# B&R Automation Studio project ProjectOrionBms
Automation Studio 4.12.6.106; technology packages: mapp 5.24.1, mappView 5.24.1

## Configuration Config1

### Task classes (Cpu.sw)
```
Cyclic#1:
  INS <- INS.INS.prg
Cyclic#2:
  AMS_CAN <- AMS_and_Shunt.CAN.AMS_CAN.prg
  INV_CAN <- Inverters.CAN.CAN.prg
Cyclic#3:
  INV_CTRL <- Inverters.Control.Control.prg
Cyclic#4:
  INV_SM <- Inverters.Inv_statemachine.Inv_statemachine.prg
  SENSORS <- Sensors.Sensors.prg
  ACTUATORS <- Actuators.Output.prg
  DASHBOARD <- Dashboard.Dashboard.prg
  COOLING <- CoolingSystem.COOLING.prg
Cyclic#5:
  Simulation <- Inverters.Simulation.Simulation.prg [disabled]
  AMS_CTRL <- AMS_and_Shunt.AMS.prg
  SC <- SC.SafetyChain.prg
  SM <- SM.StateMachine.prg
  SENSOR_NET <- SensorNet.globalSensorNet.prg [disabled]
  ALARM_MAN <- Misc.AlarmManagement.AlarmManagement.prg
Cyclic#6:
  sampleST <- Misc.DataLogging.sampleST.prg [disabled]
  DATALOG <- Misc.DataLogging.DataLog.prg
Binaries: TCData, udbdef, mvLoader, arsvcreg, OpcUaMap, ashwac, Role, ashwd, arconfig, sysconf, iomap, User, asfw, Config_1, Config, Config_2, Config_3, Acp10map, acp10cfg
Libraries: runtime, astime, standard, operator, AsIecCon, AsIODiag, brsystem, asstring, ArCan, brdkSIM, brdkUSB, AsIO, AsBrStr, sys_lib, FileIO, AsUSB, DataObj, brdkSTR, MpAlarmX, MpBase, MpData, NcGlobal, MpRecipe, sduVikings, MTTypes, dvframe, MTFilter, areventlog
```

### Config.mpalarmxcore - X90CP174_48_00/mappServices/Config.mpalarmxcore
```
Element gAlarmXCore (Type=mpalarmxcore)
  mapp.AlarmX.Core.Configuration:
    [0]:
      Name = steeringAngleSensorDisconnected
      Message = Steering angle sensor disconnected
      Behavior = LevelMonitoring
        Acknowledge = 0
        Monitoring:
          MonitoredPV = ::gSteeringAngle.status.disconnected
          HighLimitEnable = Static
            Limit = 0.5
    [1]:
      Name = steeringAngleOutOfRange
      Message = Steering angle sensor values out of range
      Behavior = LevelMonitoring
        Acknowledge = 0
        Monitoring:
          MonitoredPV = ::gSteeringAngle.status.errorOutOfRange
          LowLimitEnable = Static
          HighLimitEnable = Static
            Limit = 0.5
    [2]:
      Name = brakePressureRearOutOfRange
      Message = Brake pressure rear {&LimitText}
      Behavior = LevelMonitoring
        Acknowledge = 0
        Monitoring:
          MonitoredPV = ::gBraking.inputs.ai_brakePressureRear
          LowLimitEnable = Dynamic
            LimitPV = ::SENSORS:brakingPedalConstants.rearWarningLimitMin
            LimitText = under low limit. 
            LowLowLimitEnable = Dynamic
              LimitPV = ::SENSORS:brakingPedalConstants.rearWarningLimitMinMin
              LimitText = under low low limit. 
          HighLimitEnable = Dynamic
            LimitPV = ::SENSORS:brakingPedalConstants.rearWarningLimitMax
            LimitText = over high limit. 
            HighHighLimitEnable = Dynamic
              LimitPV = ::SENSORS:brakingPedalConstants.rearWarningLimitMaxMax
              LimitText = over high high limit. 
    [3]:
      Name = brakePressureFrontOutOfRange
      Message = Brake pressure front {&LimitText}
      Behavior = LevelMonitoring
        Acknowledge = 0
        Monitoring:
          MonitoredPV = ::gBraking.inputs.ai_brakePressureFront
          LowLimitEnable = Dynamic
            LimitPV = ::SENSORS:brakingPedalConstants.frontWarningLimitMin
            LimitText = under low limit.
            LowLowLimitEnable = Dynamic
              LimitPV = ::SENSORS:brakingPedalConstants.frontWarningLimitMinMin
              LimitText = under low low limit.
          HighLimitEnable = Dynamic
            LimitPV = ::SENSORS:brakingPedalConstants.frontWarningLimitMax
            LimitText = over high limit.
            HighHighLimitEnable = Dynamic
              LimitPV = ::SENSORS:brakingPedalConstants.frontWarningLimitMaxMax
              LimitText = over high high limit.
    [4]:
      Name = torquePedalError1
      Message = Torque pedal sensor 1 out of range
      Behavior = LevelMonitoring
        Acknowledge = 0
        Monitoring:
          MonitoredPV = ::gTorqueSensor.inputs.torque1
          LowLimitEnable = Dynamic
            LimitPV = ::SENSORS:torquePedalConstants.lowLimit1
          HighLimitEnable = Dynamic
            LimitPV = ::SENSORS:torquePedalConstants..highLimit1
    [5]:
      Name = torquePedalError2
      Message = Torque pedal sensor 2 out of range
      Behavior = LevelMonitoring
        Acknowledge = 0
        Monitoring:
          MonitoredPV = ::gTorqueSensor.inputs.torque2
          LowLimitEnable = Dynamic
            LimitPV = ::SENSORS:torquePedalConstants.lowLimit2
          HighLimitEnable = Dynamic
            LimitPV = ::SENSORS:torquePedalConstants.highLimit2
    [6]:
      Name = PowerLimitWarning_fix
      Message = Warning! Power usage close to limit
      Behavior = LevelMonitoring
        Recording:
          InactiveToActive = FALSE
          UnacknowledgedToAcknowledged = FALSE
        Monitoring:
          MonitoredPV = ::gShunt.data.actPowerKW
          Exclusive = FALSE
          HighLimitEnable = Dynamic
            LimitPV = 
            LimitText = Warning! Power limit high
    [7]:
      Name = PowerLimitError_fix
      Message = Error! Power limit exceeded!
      Behavior = LevelMonitoring
        Recording:
          InactiveToActive = FALSE
          UnacknowledgedToAcknowledged = FALSE
        Monitoring:
          MonitoredPV = ::gShunt.data.actPowerKW
          HighLimitEnable = Dynamic
            LimitPV = 
            LimitText = 
    [8]:
      Name = coolingSystemManual
      Message = Cooling system on manual mode
      Behavior = LevelMonitoring
        Acknowledge = 0
        ReactionUntilAcknowledged = FALSE
        Recording:
          InactiveToActive = FALSE
          UnacknowledgedToAcknowledged = FALSE
        Monitoring:
          MonitoredPV = ::gCooling[0].cmd.manualMode
          HighLimitEnable = Static
            Limit = 0.1
    [9]:
      Name = stateChangeTimeout
      Message = State Machine never received confirmation and had a timeout
      Behavior = LevelMonitoring
        Recording:
          InactiveToActive = FALSE
          UnacknowledgedToAcknowledged = FALSE
        Monitoring:
          MonitoredPV = ::gStateMachine.status.stateChangeTimeout
          HighLimitEnable = Static
            Limit = 0.5
    [10]:
      Name = tractionControlDisabled
      Message = Traction Control not enabled
      Behavior = LevelMonitoring
        Acknowledge = 0
        ReactionUntilAcknowledged = FALSE
        Recording:
          InactiveToActive = FALSE
          UnacknowledgedToAcknowledged = FALSE
        Monitoring:
          MonitoredPV = ::gInverters.cmd.enableTractionControl
          LowLimitEnable = Static
            Limit = 0.5
    [11]:
      Name = torqueVectoringDisabled
      Message = Torque Vectoring not enabled
      Behavior = LevelMonitoring
        Acknowledge = 0
        ReactionUntilAcknowledged = FALSE
        Recording:
          InactiveToActive = FALSE
          UnacknowledgedToAcknowledged = FALSE
        Monitoring:
          MonitoredPV = ::gInverters.cmd.enableTorqueVectoring
          LowLimitEnable = Static
            Limit = 0.5
    [12]:
      Name = powerLimiterDisabled
      Message = Power Limiter not enabled
      Behavior = LevelMonitoring
        Acknowledge = 0
        Monitoring:
          MonitoredPV = ::gInverters.cmd.enablePowerLimiter
          LowLimitEnable = Static
            Limit = 0.5
    [13]:
      Name = regenBrakingDisabled
      Message = Regenerative Braking not enabled
      Behavior = LevelMonitoring
        Acknowledge = 0
        Monitoring:
          MonitoredPV = ::gInverters.cmd.enableRegenerativeBraking
          LowLimitEnable = Static
            Limit = 0.5
    [14]:
      Name = inverter1disabled
      Message = Inverter 1 disabled
      Behavior = LevelMonitoring
        Acknowledge = 0
        Monitoring:
          MonitoredPV = ::gInverters.inverter[0].status.inverterEnabled
          LowLimitEnable = Static
            Limit = 0.5
    [15]:
      Name = inverter2disabled
      Message = Inverter 2 disabled
      Behavior = LevelMonitoring
        Acknowledge = 0
        Monitoring:
          MonitoredPV = ::gInverters.inverter[1].status.inverterEnabled
          LowLimitEnable = Static
            Limit = 0.5
    [16]:
      Name = inverter3disabled
      Message = Inverter 3 disabled
      Behavior = LevelMonitoring
        Acknowledge = 0
        Monitoring:
          MonitoredPV = ::gInverters.inverter[2].status.inverterEnabled
          LowLimitEnable = Static
            Limit = 0.5
    [17]:
      Name = inverter4disabled
      Message = Inverter 4 disabled
      Behavior = LevelMonitoring
        Acknowledge = 0
        Monitoring:
          MonitoredPV = ::gInverters.inverter[3].status.inverterEnabled
          LowLimitEnable = Static
            Limit = 0.5
    [18]:
      Name = torqueLimiting
      Message = Torque Limiting is active
      Behavior = LevelMonitoring
        Acknowledge = 0
        Recording:
          InactiveToActive = FALSE
          UnacknowledgedToAcknowledged = FALSE
        Monitoring:
          MonitoredPV = ::gInverters.cmd.enableTorqueLimiter
          HighLimitEnable = Static
            Limit = 0.5
    [19]:
      Name = inverter1ErrorDiagnostics
      Message = Inverter 1 - Error {&inverter1ErrorDiag}
      Behavior = LevelMonitoring
        Monitoring:
          MonitoredPV = ::gInverters.inverter[0].inputs.com_errorDiagnostics
          HighLimitEnable = Static
            Limit = 0.5
    [20]:
      Name = inverter2ErrorDiagnostics
      Message = Inverter 2 - Error {&inverter2ErrorDiag}
      Behavior = LevelMonitoring
        Monitoring:
          MonitoredPV = ::gInverters.inverter[1].inputs.com_errorDiagnostics
          HighLimitEnable = Static
            Limit = 0.5
    [21]:
      Name = inverter3ErrorDiagnostics
      Message = Inverter 3 - Error {&inverter3ErrorDiag}
      Behavior = LevelMonitoring
        Monitoring:
          MonitoredPV = ::gInverters.inverter[2].inputs.com_errorDiagnostics
          HighLimitEnable = Static
            Limit = 0.5
    [22]:
      Name = inverter4ErrorDiagnostics
      Message = Inverter 4 - Error {&inverter4ErrorDiag}
      Behavior = LevelMonitoring
        Monitoring:
          MonitoredPV = ::gInverters.inverter[3].inputs.com_errorDiagnostics
          HighLimitEnable = Static
            Limit = 0.5
    [23]:
      Name = amsUnderVoltage
      Message = AMS Error - Cell voltage too low
      Behavior = LevelMonitoring
        Monitoring:
          MonitoredPV = ::gAMS.status.error.lowVoltage
          HighLimitEnable = Static
            Limit = 0.5
    [24]:
      Name = amsOverVoltage
      Message = AMS Error - Cell voltage too high
      Behavior = LevelMonitoring
        Monitoring:
          MonitoredPV = ::gAMS.status.error.highVoltage
          HighLimitEnable = Static
            Limit = 0.5
    [25]:
      Name = amsUnderTemperature
      Message = AMS Error - Cell temperature too low
      Behavior = LevelMonitoring
        Monitoring:
          MonitoredPV = ::gAMS.status.error.lowTemp
          HighLimitEnable = Static
            Limit = 0.5
    [26]:
      Name = amsOverTemperature
      Message = AMS Error - Cell temperature too high
      Behavior = LevelMonitoring
        Monitoring:
          MonitoredPV = ::gAMS.status.error.highTemp
          HighLimitEnable = Static
            Limit = 0.5
    [27]:
      Name = amsCommunicationErrorLTC
      Message = AMS Error - LTC6813 communication error
      Behavior = LevelMonitoring
        Monitoring:
          MonitoredPV = ::gAMS.status.error.ltc6813Com
          HighLimitEnable = Static
            Limit = 0.5
    [28]:
      Name = amsCommunicationErrorShunt
      Message = AMS Error - Shunt communication error
      Behavior = LevelMonitoring
        Monitoring:
          MonitoredPV = ::gAMS.status.error.shuntCom
          HighLimitEnable = Static
            Limit = 0.5
    [29]:
      Name = amsOpenSc
      Message = AMS Error - Unable to open safety circuit
      Behavior = LevelMonitoring
        Monitoring:
          MonitoredPV = ::gAMS.status.error.openSc
          HighLimitEnable = Static
            Limit = 0.5
    [30]:
      Name = amsCloseSc
      Message = AMS Error - Unable to close safety circuit
      Behavior = LevelMonitoring
        Monitoring:
          MonitoredPV = ::gAMS.status.error.closeSc
          HighLimitEnable = Static
            Limit = 0.5
    [31]:
      Name = amsOpenAirMinusError
      Message = AMS Error - 
Unable to open AIR- relay
      Behavior = LevelMonitoring
        Monitoring:
          MonitoredPV = ::gAMS.status.error.openAirMinus
          HighLimitEnable = Static
            Limit = 0.5
    [32]:
      Name = amsCloseAirMinusError
      Message = AMS Error - Unable to close AIR- relay
      Behavior = LevelMonitoring
        Monitoring:
          MonitoredPV = ::gAMS.status.error.closeAirMinus
          HighLimitEnable = Static
            Limit = 0.5
    [33]:
      Name = amsOpenAirPlusError
      Message = AMS Error - Unable to open AIR+ relay



      Behavior = LevelMonitoring
        Monitoring:
          MonitoredPV = ::gAMS.status.error.openAirPlus
          HighLimitEnable = Static
            Limit = 0.5
    [34]:
      Name = amsCloseAirPlusError
      Message = AMS Error - 
Unable to close AIR+ relay
      Behavior = LevelMonitoring
        Monitoring:
          MonitoredPV = ::gAMS.status.error.closeAirPlus
          HighLimitEnable = Static
            Limit = 0.5
    [35]:
      Name = amsOpenPreError
      Message = AMS Error - 
Unable to open precharge relay
      Behavior = LevelMonitoring
        Monitoring:
          MonitoredPV = ::gAMS.status.error.openPrePlus
          HighLimitEnable = Static
            Limit = 0.5
    [36]:
      Name = amsClosePreError
      Message = AMS Error - Unable to close precharge relay
      Behavior = LevelMonitoring
        Monitoring:
          MonitoredPV = ::gAMS.status.error.closePrePlus
          HighLimitEnable = Static
            Limit = 0.5
    [37]:
      Name = amsPrechargeTimeout
      Message = AMS Error - Precharge timeout
      Behavior = LevelMonitoring
        Monitoring:
          MonitoredPV = ::gAMS.status.error.preTimeout
          HighLimitEnable = Static
            Limit = 0.5
    [38]:
      Name = amsUnexpectedChargingRate
      Message = AMS Error - Unexpected Charge Rate
      Behavior = LevelMonitoring
        Monitoring:
          MonitoredPV = ::gAMS.status.error.unexpectedChargeRate
          HighLimitEnable = Static
            Limit = 0.5
    [39]:
      Name = amsUnexpectedTsCurrent
      Message = AMS Error - Unexpected TS Current
      Behavior = LevelMonitoring
        Monitoring:
          MonitoredPV = ::gAMS.status.error.unexpectedTsCurrent
          HighLimitEnable = Static
            Limit = 0.5
    [40]:
      Name = amsBankCountMismatch
      Message = AMS Error - The specified bank count from the Car does not match the meassured cells by the AMS
      Behavior = LevelMonitoring
        Monitoring:
          MonitoredPV = ::gAMS.status.error.bankCountMismatch
          HighLimitEnable = Static
            Limit = 0.5
    [41]:
      Name = amsScBroken
      Message = AMS Error - SC Broken
      Behavior = LevelMonitoring
        Monitoring:
          MonitoredPV = ::gAMS.status.error.scBroken
          HighLimitEnable = Static
            Limit = 0.5
    [42]:
      Name = amsUnfitChargingVoltage
      Message = AMS Error - Unfit Charge Voltage
      Behavior = LevelMonitoring
        Monitoring:
          MonitoredPV = ::gAMS.status.error.unexpectedChargeRate
          HighLimitEnable = Static
            Limit = 0.5
    [43]:
      Name = amsMonitorError
      Message = AMS Error - Monitor Error
      Behavior = LevelMonitoring
        Monitoring:
          MonitoredPV = ::gAMS.status.error.monitorError
          HighLimitEnable = Static
            Limit = 0.5
    [44]:
      Name = amsRelayFailed
      Message = AMS Error - Relay Failed
      Behavior = LevelMonitoring
        Monitoring:
          MonitoredPV = ::gAMS.status.error.relayFailed
          HighLimitEnable = Static
            Limit = 0.5
    [45]:
      Name = chargingCurrentWarning_fix
      Message = Charging Current Warning
      Behavior = LevelMonitoring
        Monitoring:
          MonitoredPV = 
          HighLimitEnable = Static
            Limit = 0.5
    [46]:
      Name = dashboardDisconnection
      Message = Dashboard Error - Disconnected
      Behavior = LevelMonitoring
        Acknowledge = 0
        Monitoring:
          MonitoredPV = ::gDashboard.status.DashboardDisconnected
          HighLimitEnable = Static
            Limit = 0.5
    [47]:
      Name = AMSDisconnection
      Message = AMS Error - Disconnected
      Behavior = LevelMonitoring
        Acknowledge = 0
        Monitoring:
          MonitoredPV = gAMS.status.disconnected
          HighLimitEnable = Static
            Limit = 0.5
    [48]:
      Name = RTDSDisconnection
      Message = RTDS Error - Disconnected
      Behavior = LevelMonitoring
        Acknowledge = 0
        Monitoring:
          MonitoredPV = gRTDS.status.RTDS_Disconnected
          HighLimitEnable = Static
            Limit = 0.5
    [49]:
      Name = Pump1Disconnection
      Message = Pump 1 Error - Disconnected
      Behavior = LevelMonitoring
        Acknowledge = 0
        Monitoring:
          MonitoredPV = gCooling.status.error[0]
          HighLimitEnable = Static
            Limit = 0.5
    [50]:
      Name = Pump2Disconnection
      Message = Pump 2 Error - Disconnected
      Behavior = LevelMonitoring
        Acknowledge = 0
        Monitoring:
          MonitoredPV = gCooling.status.error[1]
          HighLimitEnable = Static
            Limit = 0.5
    [51]:
      Name = LowVoltageBatteryLow
      Message = Warning! LV battery low 
      Behavior = LevelMonitoring
        Acknowledge = 0
        Monitoring:
          MonitoredPV = gLowVoltageBattery.status.empty
          HighLimitEnable = Static
            Limit = 0.5
    [52]:
      Name = inverter1Disconnected
      Message = Inverter 1 disconnected
      Behavior = LevelMonitoring
        Monitoring:
          MonitoredPV = ::gInverters.inverter[0].status.inverterDisconnected
          HighLimitEnable = Static
            Limit = 0.5
    [53]:
      Name = inverter2Disconnected
      Message = Inverter 2 disconnected
      Behavior = LevelMonitoring
        Acknowledge = 0
        Monitoring:
          MonitoredPV = ::gInverters.inverter[1].status.inverterDisconnected
          HighLimitEnable = Static
            Limit = 0.5
    [54]:
      Name = inverter3Disconnected
      Message = Inverter 3 disconnected
      Behavior = LevelMonitoring
        Acknowledge = 0
        Monitoring:
          MonitoredPV = ::gInverters.inverter[2].status.inverterDisconnected
          HighLimitEnable = Static
            Limit = 0.5
    [55]:
      Name = inverter4Disconnected
      Message = Inverter 4 disconnected
      Behavior = LevelMonitoring
        Acknowledge = 0
        Monitoring:
          MonitoredPV = ::gInverters.inverter[3].status.inverterDisconnected
          HighLimitEnable = Static
            Limit = 0.5
    [56]:
      Name = dataloggingInactive
      Message = Datalogging disabled
      Behavior = LevelMonitoring
        Monitoring:
          MonitoredPV = ::gDataLogging.status.dataloggingActive
          HighLimitEnable = Static
            Limit = 0.5
    [57]:
      Name = torquePedalPlausibilityError
      Message = Torque Pedal Plausibility Error
      Behavior = LevelMonitoring
        Monitoring:
          MonitoredPV = ::gTorqueSensor.status.plausibilityError
          HighLimitEnable = Static
            Limit = 0.5
    [58]:
      Name = shuntDisconnection
      Message = Shunt disconnected
      Behavior = LevelMonitoring
        Monitoring:
          MonitoredPV = ::gShunt.status.disconnected
          HighLimitEnable = Static
            Limit = 0.5
    [59]:
      Name = scBroken
      Message = SC Error - {&scErrorString}
      Behavior = DiscreteValueMonitoring
        ReactionUntilAcknowledged = FALSE
        Monitoring:
          MonitoredPV = ::gSafetyChain.status.scErrorIndex
          TriggerValues:
            [0] = 1
            [1] = 2
            [2] = 3
            [3] = 4
            [4] = 5
            [5] = 6
            [6] = 7
            [7] = 8
            [8] = 9
            [9] = 10
            [10] = 11
            [11] = 12
            [12] = 13
            [13] = 14
            [14] = 15
            [15] = 16
            [16] = 17
            [17] = 18
            [18] = 19
            [19] = 20
            [20] = 21
            [21] = 22
            [22] = 
    [60]:
      Name = inverterHighTemperature
      Message = Warning! Inverters are getting hot
      Behavior = LevelMonitoring
        Monitoring:
          MonitoredPV = ::gCooling.status.warningInverterHighTemp
          HighLimitEnable = Static
            Limit = 0.5
    [61]:
      Name = motorHighTemperature
      Message = Warning! Motors are getting hot
      Behavior = LevelMonitoring
        Monitoring:
          MonitoredPV = ::gCooling.status.warningMotorHighTemp
          HighLimitEnable = Static
            Limit = 0.5
    [62]:
      Name = orionBmsCommTimeout
      Message = Error! No Communication with Orion BMS
      Behavior = LevelMonitoring
        Monitoring:
          MonitoredPV = ::gORION.status.commTimeout
          HighLimitEnable = Static
            Limit = 0.5
  mapp.AlarmX.Core.Snippets:
    [0]:
      Key = inverter1ErrorDiag
      Value:
        PV = ::gInverters.inverter[0].inputs.com_errorDiagnostics
    [1]:
      Key = inverter2ErrorDiag
      Value:
        PV = ::gInverters.inverter[1].inputs.com_errorDiagnostics
    [2]:
      Key = inverter3ErrorDiag
      Value:
        PV = ::gInverters.inverter[2].inputs.com_errorDiagnostics
    [3]:
      Key = inverter4ErrorDiag
      Value:
        PV = ::gInverters.inverter[3].inputs.com_errorDiagnostics
    [4]:
      Key = scErrorString
      Value:
        PV = ::gSafetyChain.status.scErrorString
```

### Config_2.mpdatarecorder - X90CP174_48_00/mappServices/Config_2.mpdatarecorder
```
Element gDataRecorder (Type=mpdatarecorder)
```

### Config_3.mprecipexml - X90CP174_48_00/mappServices/Config_3.mprecipexml
```
Element gRecipeXml (Type=mprecipexml)
```

## Logical view

Binary libraries used (declarations not repeated): MpData 5.24.1

### Program Logical/Actuators/Output

#### Main.st
```iecst
PROGRAM _INIT
	(* Initialize outputs *)
	RtdsInit;

END_PROGRAM

PROGRAM _CYCLIC
	// Handle Ready-To-Drive-Sounds
	Rtds;

END_PROGRAM

PROGRAM _EXIT
	(* Insert code here *)

END_PROGRAM
```

### globalORION.typ
```iecst
TYPE
	gORION_state_ENUM :
		(
		INIT := 0,
		IDLE := 10,
		ENABLING_SC := 20,
		SC_ENABLED := 30,
		PRECHARGING := 40,
		PRECHARGING_DONE := 50,
		DRIVE_PRECHARGE_ACTIVE := 60,
		DRIVE := 70,
		ABORT := 80,
		ERROR := 90
		);
	gORION_relays_typ : 	STRUCT
		sdcEnable : BOOL;
		precharge : BOOL;
		airMinus : BOOL;
		airPlus : BOOL;
	END_STRUCT;
	gORION_typ : 	STRUCT
		state : gORION_state_ENUM;
		cmd : gORION_cmd_typ;
		status : gORION_status_typ;
		relays : gORION_relays_typ;
		data : gORION_data_typ;
	END_STRUCT;
	gORION_cmd_typ : 	STRUCT
		placeholder : USINT;
	END_STRUCT;
	gORION_status_typ : 	STRUCT
		sdcEnabled : BOOL;
		commTimeout : BOOL;
	END_STRUCT;
	gORION_data_typ : 	STRUCT
		packVoltage : REAL;
		prechargeLevel : REAL;
		carVoltage : REAL;
		maxPrechargeCurrent : REAL;
		chargeCurrent : REAL;
		outputCurrent : REAL;
		TON_counter : TON;
		CCL_KW : REAL;
		CCL : INT;
		DCL_KW : REAL;
		DCL : INT;
		rollingCounterOld : USINT;
		rollingCounter : USINT;
		packPower : REAL;
	END_STRUCT;
END_TYPE
```

### Program Logical/AMS_and_Shunt/AMS

#### Variables.var
```iecst
VAR
	k : UINT;
	j : USINT;
	i : UINT;
	tmpTemperatureMax : REAL;
	tmpTemperatureMin : REAL;
	tmpVoltageMax : REAL;
	tmpVoltageMin : REAL;
	tmpVoltage : REAL;
	TON_historySoc : TON;
	TON_historyCurrent : TON;
	TON_historyVoltage : TON;
	TON_historyPower : TON;
	powerHistoryInverval : TIME;
	currentHistoryInverval : TIME;
	voltageHistoryInverval : TIME;
	socHistoryInverval : TIME;
	powerWarningLimit : REAL;
	constant : constant_typ;
	CMD_ABORT : USINT := 0;
	CMD_ENABLE_SC : USINT := 1;
	CMD_ENABLE_TS : USINT := 2;
	CMD_ENABLE_DRIVE : USINT := 3;
	CMD_SET_BANK_COUNT : USINT := 5;
	CMD_SYNC_TIME : USINT := 6;
	inrushCurrentDetected : BOOL;
END_VAR
```

#### Main.st
```iecst
PROGRAM _INIT

	gAMS.data.outputCurrent := 0;
	gAMS.data.stateOfCharge := 0;
//	gAMS.data.totalPower 	:= 0;
//	gAMS.data.totalPowerMax := 0;  // Reset variable used to keep track of the maximum power used

	powerHistoryInverval 		:= T#10ms;
	currentHistoryInverval 		:= T#20ms;
	socHistoryInverval			:= T#500ms;
	voltageHistoryInverval  	:= T#100ms;
	gORION.data.TON_counter.PT	:= T#1s;

	constant.fullBatteryCapacityAh  := 12.5;
	constant.fullBatteryCapacitykWh := 6.475;

	constant.chargingCurrentMax := 12.5;
	gAMS.cmd.chargingPrescalerAmp := constant.chargingCurrentMax;

	gAMS.cmd.bankCount := 5;

	errorsInit_action;

END_PROGRAM

PROGRAM _CYCLIC

	states;
	orionErrorAction;
	error_action;

	gAMS.data.chargeCurrent := - gAMS.data.outputCurrent;

//	gAMS.data.batteryVoltage := gAMS.status.bank[0].bankVoltage + gAMS.status.bank[1].bankVoltage +
//								gAMS.status.bank[2].bankVoltage + gAMS.status.bank[3].bankVoltage +
//								gAMS.status.bank[4].bankVoltage;

	gAMS.cmd.chargingPrescalerPercent := LIMIT(0, REAL_TO_USINT((gAMS.cmd.chargingPrescalerAmp / constant.chargingCurrentMax) * 100), 100);

	powerMonitoring;

	(* Determine if AMS has an error or not *)
	gAMS.status.ok 	 := (NOT gAMS.status.disconnected) AND (NOT (gAMS.status.amsStateName = 'ERROR')) AND (NOT gAMS.status.hasError);
	gShunt.status.ok := NOT gShunt.status.disconnected;

//	gAMS.data.stateOfCharge := ((constant.fullBatteryCapacitykWh-gShunt.data.actPowerKWH) / constant.fullBatteryCapacitykWh) * 100.00;

	// Calculating the voltage of each bank
	FOR j := 0 TO BANK_COUNT-1 DO
		k := CELL_COUNT*j;
		tmpVoltage := 0;
		FOR i := 0 TO CELL_COUNT-1 DO
			// gAMS.status.bank[j].cellVoltage[i] := gAMS.status.pack.cellVoltage[i + k];
			tmpVoltage := tmpVoltage + gAMS.status.bank[j].cellVoltage[i];
		END_FOR;
		gAMS.status.bank[j].bankVoltage := tmpVoltage;
	END_FOR

	FOR j := 0 TO BANK_COUNT-1 DO
		// Max voltage
		tmpVoltageMax := 0;
		FOR i := 0 TO CELL_COUNT-1 DO
			IF gAMS.status.bank[j].cellVoltage[i] > tmpVoltageMax THEN
				tmpVoltageMax := gAMS.status.bank[j].cellVoltage[i];
			END_IF;
		END_FOR;
		gAMS.data.cellVoltageMax[j] := tmpVoltageMax;

		// Min voltage
		tmpVoltageMin := 10000;
		FOR i := 0 TO CELL_COUNT-1 DO
			IF gAMS.status.bank[j].cellVoltage[i] < tmpVoltageMin THEN
				tmpVoltageMin := gAMS.status.bank[j].cellVoltage[i];
			END_IF;
		END_FOR;
		gAMS.data.cellVoltageMin[j] := tmpVoltageMin;

		// Max temperature
		tmpTemperatureMax := 0;
		FOR i := 0 TO TEMPERATURE_COUNT-1 DO
			IF gAMS.status.bank[j].temperatures[i] > tmpTemperatureMax THEN
				tmpTemperatureMax := gAMS.status.bank[j].temperatures[i];
			END_IF;
		END_FOR;
		gAMS.data.bankTemperatureMax[j] := tmpTemperatureMax;

		// Min temperature
		tmpTemperatureMin := 10000;
		FOR i := 0 TO TEMPERATURE_COUNT-1 DO
			IF gAMS.status.bank[j].temperatures[i] < tmpTemperatureMin THEN
				tmpTemperatureMin := gAMS.status.bank[j].temperatures[i];
			END_IF;
		END_FOR;
		gAMS.data.bankTemperatureMin[j] := tmpTemperatureMin;

		// Max resistor temperature
		tmpTemperatureMax := 0;
		FOR i := 0 TO RESISTOR_COUNT-1 DO
			IF gAMS.status.bank[j].resistorTemperature[i] > tmpTemperatureMax THEN
				tmpTemperatureMax := gAMS.status.bank[j].resistorTemperature[i];
			END_IF;
		END_FOR;
		gAMS.data.bankResistorTemperatureMax[j] := tmpTemperatureMax;

		// Min temperature
		tmpTemperatureMin := 10000;
		FOR i := 0 TO RESISTOR_COUNT-1 DO
			IF gAMS.status.bank[j].resistorTemperature[i] < tmpTemperatureMin THEN
				tmpTemperatureMin := gAMS.status.bank[j].resistorTemperature[i];
			END_IF;
		END_FOR;
		gAMS.data.bankResistorTemperatureMin[j] := tmpTemperatureMin;

	END_FOR;

	history;

END_PROGRAM

PROGRAM _EXIT
	(* Insert code here *)

END_PROGRAM
```

#### powerMonitoring.st
```iecst
(* Keep track of the current power consumption and the maximum power *)
ACTION powerMonitoring:
	// Actual power
//	gAMS.data.totalPowerKW := gAMS.data.totalPower / 1000.00;

	// Maximum power
//	IF gAMS.data.totalPower > gAMS.data.totalPowerMax THEN
//		gAMS.data.totalPowerMax := gAMS.data.totalPower;
//		gAMS.data.totalPowerMaxKW := gAMS.data.totalPowerMax / 1000.00;
//	END_IF;

	IF gInverters.cmd.enablePowerLimiter THEN
//		powerWarningLimit := gInverters.data.powerLimitKW*0.9;
//		IF gAMS.data.totalPowerKW > 1 THEN
//			gAMS.status.highPowerWarning := powerWarningLimit 					<= gAMS.data.totalPowerKW;
//			gAMS.status.highPowerError   := gInverters.data.powerLimitKW 	<= gAMS.data.totalPowerKW;
//		END_IF;
	ELSE
		gAMS.status.highPowerWarning := FALSE;
		gAMS.status.highPowerError   := FALSE;
	END_IF;

END_ACTION
```

### Program Logical/AMS_and_Shunt/CAN/AMS_CAN (IEC)

#### Main.st
```iecst
PROGRAM _INIT
	(* Device *)
	deviceName 						:= 'IF9';
	(* Bus *)
	ArCanSetBaudrate_0.Baudrate 	:= 500000;
	(* Transmit *)
	ArCanSend_0.Frame.Format 		:= arCAN_11BIT;
	(* Receive *)
	ArCanReceive_0.Format 			:= arCAN_11BIT;
	ArCanReceive_0.QueueSize		:= 100;
	ArCanReceive_0.IDMask			:= arCAN_RECEIVE_ALL;

	communicationState := S_INIT;

	RX_CAN_ID_BASE 		:= 16#300;
	TX_CAN_ID_BASE 		:= 16#300;
	RX_ORION_ID_BASE	:= 16#400;
	TX_ORION_ID_BASE	:= 16#400;
	SHUNT_ID_BASE  		:= 16#500;

	NO_OF_BANKS := 4;
//	gAMS.status.error.dataFrameLost := FALSE;

END_PROGRAM

PROGRAM _CYCLIC

	CASE communicationState OF
		S_INIT:
			(* PLC is not simulated. It is run on an actual PLC *)
			IF NOT gIsSimulation THEN

				(* Configure CAN port *)
				ArCanSetBaudrate_0.DeviceName	:= deviceName;
				ArCanSetBaudrate_0.Execute 		:= TRUE;
				IF ArCanSetBaudrate_0.Done THEN
					communicationState 			:= S_INIT_TX;
				END_IF;
				IF ArCanSetBaudrate_0.Error THEN
					communicationState 			:= S_ERROR;
				END_IF;
			ELSE
				(* PLC is simulated. It is run in the simulator and no hardware is connnected *)
				communicationState 				:= S_IDLE;
			END_IF;

		S_INIT_TX: // Init Tx
			(* Configure send function block *)
			ArCanSend_0.Enable 			:= TRUE;
			ArCanSend_0.DeviceName 		:= deviceName;

			IF ArCanSend_0.Active THEN
				communicationState 		:= S_INIT_RX;
			END_IF;

			IF ArCanSend_0.Error THEN
				communicationState 		:= S_ERROR;
			END_IF;

		S_INIT_RX:	// Init Rx
			(* Configure receive function block *)
			ArCanReceive_0.Enable 		:= TRUE;
			ArCanReceive_0.DeviceName 	:= deviceName;

			IF ArCanReceive_0.Active THEN
				communicationState 		:= S_RUNNING;
			END_IF;

			IF ArCanReceive_0.Error THEN
				communicationState 		:= S_ERROR;
			END_IF

		S_RUNNING: // Running
			AMS_Send;		// Handle transmit task
			AMS_Receive;	// Handle receive task

		S_ERROR: // Error
			IF ArCanSend_0.Error THEN
				ArCanSend_0(Enable := FALSE);
				ArCanSend_0(Enable := TRUE);
			END_IF;

			IF ArCanReceive_0.Error THEN
				ArCanReceive_0(Enable := FALSE);
				ArCanReceive_0(Enable := TRUE);
			END_IF;

			IF (ArCanReceive_0.Error = FALSE) AND (ArCanSend_0.Error = FALSE) AND (ArCanSetBaudrate_0.Error = FALSE) THEN
				communicationState 		:= S_INIT;
			END_IF;
		S_IDLE: // Do nothing
	END_CASE

	IF NOT gIsSimulation THEN
		ArCanSetBaudrate_0();
		ArCanReceive_0();
		ArCanSend_0();
	END_IF;

//	gAMS.status.error.dataFrameLost := ArCanReceive_0.NumberOfLostFrames <> 0;

END_PROGRAM

PROGRAM _EXIT
	(* Insert code here *)

END_PROGRAM
```

### Program Logical/CoolingSystem/COOLING

#### Variables.var
```iecst
VAR
	COOLING_MODE_STATE : USINT := 0;
	pumpOffCurrent : UINT;
	pumpOnCurrent : UINT;
	i : USINT;
END_VAR
```

#### Main.st
```iecst
PROGRAM _INIT
	pumpOffCurrent := 1000;
	pumpOnCurrent  := 9500;
	gCooling.cmd.manualMode := FALSE;
	//gCooling.outputs.do_pump[1] := TRUE;
	FOR i := 0 TO 1 DO
		gCooling.outputs.do_pump[i] 	:= TRUE;
		gCooling.outputs.do_fan[i] 		:= TRUE;
		//gCooling.outputs.do_pump[i] 	:= FALSE;
		//gCooling.outputs.do_fan[i] 		:= FALSE;
	END_FOR

	gCooling.status.warningHighTemperature := FALSE;

	gCooling.cmd.inverterMaxTemp 	:= 60.0;
	gCooling.cmd.motorMaxTemp 		:= 100.0;
END_PROGRAM

PROGRAM _CYCLIC

	CASE COOLING_MODE_STATE OF
		0: // AUTO MODE
			IF gDashboard.inputs.di_button2 AND (gInverters.inverter[0].data.actualVelocityKmh = 0) THEN
	  			COOLING_MODE_STATE := 10;
			END_IF;
			IF gStateMachine.status.state = STATE_DRIVE THEN
				COOLING_MODE_STATE := 10;
			END_IF;
		10: // going to MANUAL MODE
			IF NOT gDashboard.inputs.di_button2 THEN
				gCooling.cmd.manualMode := TRUE;
				gCooling.outputs.do_pump[1] := TRUE;
				COOLING_MODE_STATE := 20;
			END_IF;

		20: // MANUAL MODE
			IF gDashboard.inputs.di_button2 AND (gInverters.inverter[0].data.actualVelocityKmh = 0) THEN
				COOLING_MODE_STATE := 30;
			END_IF;

		30:
			IF NOT gDashboard.inputs.di_button2 THEN
				gCooling.cmd.manualMode := FALSE;
				gCooling.outputs.do_pump[1] := FALSE;
				COOLING_MODE_STATE := 0;
			END_IF
	END_CASE;

	(* Convert analog temperature inputs to temperatures in degrees *)
	FOR i := 0 TO 1 DO
		(* Cooling System Temperature approximated via 4th order polynomium *)
		gCooling.data.coolingSysTemp[i] := EXPT(gCooling.inputs.ai_coolingTemp[i],2) + 0.004914 * gCooling.inputs.ai_coolingTemp[i] - 44.62;
	END_FOR

	// If cooling system is not in manual mode (its in automatic mode)
	IF NOT gCooling.cmd.manualMode THEN
		FOR i := 0 TO 1 DO
			//IF gCooling.outputs.do_pump[i] THEN
				//IF INT_TO_UINT(gCooling.inputs.im_pumpCurrent[i]) < pumpOffCurrent THEN
					// No current is being drawn
				//	gCooling.status.pumpState[i] := PUMP_STATE_NOT_CONNECTED;
				//ELSIF INT_TO_UINT(gCooling.inputs.im_pumpCurrent[i]) > pumpOffCurrent AND INT_TO_UINT(gCooling.inputs.im_pumpCurrent[i]) < pumpOnCurrent THEN
					// Not enough current is being drawn
				//	gCooling.status.pumpState[i] := PUMP_STATE_NO_WATER;
				//ELSE
			// Normal amount of current is being drawn
				IF gStateMachine.status.state = STATE_TRACTIVE THEN
					gCooling.status.pumpState[i] := PUMP_STATE_OK;
				ELSE
					gCooling.status.pumpState[i] := PUMP_STATE_NO_WATER; // Just to turn off when not in tractive
				END_IF;

				// Check if there is an error on the pump. If the pump state is not OK there is an error
				gCooling.status.pumpError[i] := gCooling.status.pumpState[i] <> PUMP_STATE_OK;

				// If there is an error turn OFF the pump. Otherwise keep it ON
				gCooling.outputs.do_pump[i] := NOT gCooling.status.pumpError[i];

			//END_IF

		END_FOR
	END_IF;

	// Enable fan when in STATE_DRIVE
	FOR i := 0 TO 1 DO
		gCooling.outputs.do_fan[i] := gStateMachine.status.state = STATE_DRIVE;
	END_FOR;

	// Evaluate if inverter or motors have high temperature errors
	gCooling.status.warningInverterHighTemp := MAX(gInverters.inverter[0].data.tempInverter, gInverters.inverter[1].data.tempInverter, gInverters.inverter[2].data.tempInverter, gInverters.inverter[3].data.tempInverter) > gCooling.cmd.inverterMaxTemp;
	gCooling.status.warningMotorHighTemp 	:= MAX(gInverters.inverter[0].data.tempMotor   , gInverters.inverter[1].data.tempMotor,    gInverters.inverter[2].data.tempMotor,    gInverters.inverter[3].data.tempMotor)    > gCooling.cmd.motorMaxTemp;

	// Evaluate if the cooling system is working properly.
	gCooling.status.ok := NOT gCooling.status.pumpError[0] AND NOT gCooling.status.pumpError[1];

	// Evaluate if the cooling system sees any temperature higher than allowed
	gCooling.status.warningHighTemperature := gCooling.status.warningInverterHighTemp OR gCooling.status.warningMotorHighTemp;
END_PROGRAM

PROGRAM _EXIT
	(* Insert code here *)

END_PROGRAM
```

### globalDashboard.var
```iecst
VAR
	gDashboard : gDashboard_typ;
END_VAR
```

### Program Logical/Dashboard/Dashboard/ledControl

#### ledDV.st
```iecst
(* Control the DV LED *)
ACTION ledDV:
	IF gStateMachine.status.state = STATE_INITIALIZE THEN
		gDashboard.outputs.do_ledDV := TRUE;
	ELSE
		gDashboard.outputs.do_ledDV := FALSE;
	END_IF;
END_ACTION
```

#### ledEBS.st
```iecst
(* Control the EBS LED *)
ACTION ledEBS:
	IF gStateMachine.status.state = STATE_INITIALIZE THEN
		gDashboard.outputs.do_ledEBS := TRUE;
	ELSE
		gDashboard.outputs.do_ledEBS := FALSE;
	END_IF;
END_ACTION
```

#### ledIMD.st
```iecst
(* Control the IMD LED *)
ACTION ledIMD:
	IF gStateMachine.status.state = STATE_INITIALIZE THEN
		gDashboard.outputs.do_ledIMD := TRUE;
	ELSE
		gDashboard.outputs.do_ledIMD := gAMS.status.error.imdError;
	END_IF;
END_ACTION
```

#### ledLV.st
```iecst
(* Control the LV LED *)
ACTION ledLV:

	IF gStateMachine.status.state = STATE_INITIALIZE THEN
		gDashboard.outputs.do_ledLV := FALSE;

	ELSE
		IF gLowVoltageBattery.status.empty THEN
			gDashboard.outputs.do_ledLV := TRUE;
		ELSE
			gDashboard.outputs.do_ledLV := FALSE;
		END_IF;

	END_IF;

END_ACTION
```

#### ledREADY.st
```iecst
(* Control the READY LED *)
ACTION ledREADY:
	IF gStateMachine.status.state = STATE_INITIALIZE THEN
		gDashboard.outputs.do_ledREADY := READY_ON;
	ELSE
		IF gStateMachine.status.state = STATE_DRIVE THEN
			gDashboard.outputs.do_ledREADY := READY_ON;
		ELSIF gStateMachine.status.readyForStateDrive THEN
			gDashboard.outputs.do_ledREADY := READY_FAST_BLINK;
		ELSIF gStateMachine.status.state = STATE_TRACTIVE THEN
			gDashboard.outputs.do_ledREADY := READY_SLOW_BLINK;
		ELSE
			gDashboard.outputs.do_ledREADY := READY_OFF;
		END_IF
	END_IF

	// Slow blink: State = TRACTIVE
	// Fast blink: State = TRACTIVE & gBraking.status.softBraking = TRUE & NOT gTorqueSensor.status.criticalError
	// On = DRIVE
	// Off : Else

END_ACTION
```

### Program Logical/Dashboard/Dashboard/Receive

#### receive_messages.st
```iecst
ACTION msg_0x050:
	gDashboard.inputs.di_buttonSafety		:= ArCanReceive_0.ReceivedFrame.Data[0].0;
	gDashboard.inputs.di_buttonTractive		:= ArCanReceive_0.ReceivedFrame.Data[0].1;
	gDashboard.inputs.di_buttonDrive		:= ArCanReceive_0.ReceivedFrame.Data[0].2;
	gDashboard.inputs.di_button1			:= ArCanReceive_0.ReceivedFrame.Data[0].3;
//
//	gDashboard.inputs.di_buttonDrive		:= ArCanReceive_0.ReceivedFrame.Data[0].3;
//	gDashboard.inputs.di_button1			:= ArCanReceive_0.ReceivedFrame.Data[0].2;
//
	gDashboard.inputs.di_button2			:= ArCanReceive_0.ReceivedFrame.Data[0].4;
	gDashboard.inputs.di_button3			:= ArCanReceive_0.ReceivedFrame.Data[0].5;
	gDashboard.inputs.di_button4			:= ArCanReceive_0.ReceivedFrame.Data[0].6;
END_ACTION

ACTION msg_0x051:
	gDashboard.status.statusIndex := BYTE_TO_USINT(ArCanReceive_0.ReceivedFrame.Data[0]);
END_ACTION

ACTION msg_0x052:
	(* Chagne driving mission *)
	CASE BYTE_TO_USINT(ArCanReceive_0.ReceivedFrame.Data[0]) OF
		MISSION_NONE: 		  gStateMachine.status.missionIndex := MISSION_NONE;
		MISSION_ACCELERATION: gStateMachine.status.missionIndex := MISSION_ACCELERATION;
		MISSION_SKIDPAD: 	  gStateMachine.status.missionIndex := MISSION_SKIDPAD;
		MISSION_SPRINT: 	  gStateMachine.status.missionIndex := MISSION_SPRINT;
		MISSION_ENDURANCE: 	  gStateMachine.status.missionIndex := MISSION_ENDURANCE;
		MISSION_BRAKE_TEST:	  gStateMachine.status.missionIndex := MISSION_BRAKE_TEST;
		MISSION_TESTING: 	  gStateMachine.status.missionIndex := MISSION_TESTING;
		ELSE	  			  gStateMachine.status.missionIndex := MISSION_NONE;
	END_CASE;
END_ACTION
```

### send_messages.st
```iecst
(*
Protocol specifications
https://gitlab.com/sdu-vikings/X/master-controller/-/wikis/Dashboard-CAN-Protocol
*)

ACTION msg_0x000:
	ArCanSend_0.Frame.ID 		  := TX_CAN_ID_BASE + 16#000; // CAN-ID
	ArCanSend_0.Frame.DataLength  := 6; 	 // Datalength

	speed 			:=	REAL_TO_INT(  gINS.data.actLonVelocity_kmh * 10.00 );
	soc 			:=	REAL_TO_INT(  gAMS.data.stateOfCharge * 10.00 );
	maxTemperature  := 	REAL_TO_UINT(MAX(gInverters.inverter[0].data.tempMotor, gInverters.inverter[1].data.tempMotor, gInverters.inverter[2].data.tempMotor, gInverters.inverter[3].data.tempMotor) * 10.00);

	memcpy(ADR(ArCanSend_0.Frame.Data[0]), ADR( speed 			), 2);
	memcpy(ADR(ArCanSend_0.Frame.Data[2]), ADR( soc 			), 2);
	memcpy(ADR(ArCanSend_0.Frame.Data[4]), ADR( maxTemperature	), 2);

END_ACTION

ACTION msg_0x001:
	ArCanSend_0.Frame.ID 		  := TX_CAN_ID_BASE+ 16#001; // CAN-ID
	ArCanSend_0.Frame.DataLength  := 4; 	 // Datalength

	memcpy(ADR(ArCanSend_0.Frame.Data[0]), ADR( gStateMachine.status.instructionIndex 	), 1);
	memcpy(ADR(ArCanSend_0.Frame.Data[1]), ADR( gStateMachine.status.state 				), 1);
	ArCanSend_0.Frame.Data[2].0 := gDashboard.outputs.com_error_Datalog;
	ArCanSend_0.Frame.Data[2].1 := gDashboard.outputs.com_error_SC;
	ArCanSend_0.Frame.Data[2].2 := gDashboard.outputs.com_error_Shunt;
	ArCanSend_0.Frame.Data[2].3 := gDashboard.outputs.com_error_AMS;
	ArCanSend_0.Frame.Data[2].4 := gDashboard.outputs.com_error_Dashboard;
	ArCanSend_0.Frame.Data[2].5 := gDashboard.outputs.com_error_3rd_Inv;
	ArCanSend_0.Frame.Data[2].6 := gDashboard.outputs.com_error_2nd_Inv;
	ArCanSend_0.Frame.Data[2].7 := gDashboard.outputs.com_error_1st_Inv;
	ArCanSend_0.Frame.Data[3].0 := gDashboard.outputs.com_error_0_Inv;
	ArCanSend_0.Frame.Data[3].1 := gDashboard.outputs.com_error_INS;
	ArCanSend_0.Frame.Data[3].2 := gDashboard.outputs.com_error_SteeringAngle;
	ArCanSend_0.Frame.Data[3].3 := gDashboard.outputs.com_error_BreakPressure_Front;
	ArCanSend_0.Frame.Data[3].4 := gDashboard.outputs.com_error_BreakPressure_Back;
	ArCanSend_0.Frame.Data[3].5 := gDashboard.outputs.com_error_TorquePedal;
	ArCanSend_0.Frame.Data[3].6 := gDashboard.outputs.com_error_TorquePedal_Plausi;
	ArCanSend_0.Frame.Data[3].7 := gDashboard.outputs.com_error_RTDS;
	ArCanSend_0.Frame.Data[4].0 := gDashboard.outputs.com_error_Cooling;
	ArCanSend_0.Frame.Data[4].1 := gDashboard.outputs.com_error_LV;
	ArCanSend_0.Frame.Data[4].2 := gDashboard.outputs.com_error_HighTemperature;

END_ACTION

ACTION msg_0x002:
	ArCanSend_0.Frame.ID 		  := TX_CAN_ID_BASE + 16#002; // CAN-ID
	ArCanSend_0.Frame.DataLength  := 2; 	 // Datalength

	ArCanSend_0.Frame.Data[0].0 := gDashboard.outputs.do_ledIMD;
	ArCanSend_0.Frame.Data[0].1 := gDashboard.outputs.do_ledAMS;
	ArCanSend_0.Frame.Data[0].2 := gDashboard.outputs.do_ledSC.0;
	ArCanSend_0.Frame.Data[0].3 := gDashboard.outputs.do_ledSC.1;
	ArCanSend_0.Frame.Data[0].4 := gDashboard.outputs.do_ledEBS;
	ArCanSend_0.Frame.Data[0].5 := gDashboard.outputs.do_ledDV;
	ArCanSend_0.Frame.Data[0].6 := gDashboard.outputs.do_ledREADY.0;
	ArCanSend_0.Frame.Data[0].7 := gDashboard.outputs.do_ledREADY.1;
	ArCanSend_0.Frame.Data[1].0 := gDashboard.outputs.do_ledLV;

END_ACTION

ACTION msg_0x003:
	ArCanSend_0.Frame.ID 		  := TX_CAN_ID_BASE + 16#003; // CAN-ID
	ArCanSend_0.Frame.DataLength := 6; 	 // Datalength

	memcpy(ADR(ArCanSend_0.Frame.Data[0]), ADR(gStateMachine.status.missionIndex), 1);

	ArCanSend_0.Frame.Data[1].0 := gInverters.cmd.enableTorqueVectoring;
	ArCanSend_0.Frame.Data[1].1 := gInverters.cmd.enableTractionControl;
	ArCanSend_0.Frame.Data[1].2 := gInverters.cmd.enablePowerLimiter;
	ArCanSend_0.Frame.Data[1].3 := gInverters.cmd.enableTorqueLimiter;
	//	ArCanSend_0.Frame.Data[1].4 := gInverters.cmd.enableLaunchProfile;
	ArCanSend_0.Frame.Data[1].5 := gInverters.cmd.enableRegenerativeBraking;
	ArCanSend_0.Frame.Data[1].6 := gInverters.status.regenerativeBrakingAvailable;
	torqueLimitNm  				:= REAL_TO_UINT(gInverters.data.torqueSetpointGain * 10.00);
	powerLimitKW  				:= REAL_TO_UINT(gInverters.data.powerLimitKW * 10.00);

	memcpy(ADR(ArCanSend_0.Frame.Data[2]), ADR(torqueLimitNm), 2);
	memcpy(ADR(ArCanSend_0.Frame.Data[4]), ADR(powerLimitKW), 2);
END_ACTION

ACTION msg_0x004:
	ArCanSend_0.Frame.ID 		  := TX_CAN_ID_BASE + 16#004; // CAN-ID
	ArCanSend_0.Frame.DataLength := 4; 	 // Datalength

	lvBatVoltage  		:= 	REAL_TO_UINT( gLowVoltageBattery.data.voltage * 10.00 );
	estimatedRange  	:=  REAL_TO_UINT( gINS.data.distEstimated * 10.00 );

	memcpy(ADR(ArCanSend_0.Frame.Data[0]), ADR( lvBatVoltage 	), 2);
	memcpy(ADR(ArCanSend_0.Frame.Data[2]), ADR( estimatedRange  ), 2);

END_ACTION
```

### Program Logical/INS/INS

#### Main.st
```iecst
PROGRAM _INIT
	// Enable serial communication
	Receiver.Commands.open_receive := TRUE;												(*enable Receiver by default*)

	(* Range Estimation *)
	MTFilterMovingAverage_0.Enable 		 := TRUE;
	MTFilterMovingAverage_0.WindowLength := 10;
	TON_rangEstTimer.PT 				 := T#10s;

	// Get cycle time
	RTInfo_0(enable := TRUE);
	cycletime := RTInfo_0.cycle_time / 1000; //[ms]

	gINS.data.distEstimated := 0;
END_PROGRAM

PROGRAM _CYCLIC

	// If the state is any of the 3 states used for receiving and decoding data mark the INS as ok
	// Otherwise mark it as not ok
	gINS.status.ok := Receiver.step = FRM_READ OR Receiver.step = FRM_COPY_RD_DATA OR Receiver.step = FRM_RBUF;

	// Handle communication
	CASE Receiver.step OF
		FRM_WAIT:	(*--- wait for command*)

			IF Receiver.Commands.open_receive = TRUE THEN								(*command for Receiver activation*)
				Receiver.step := FRM_OPEN;
			END_IF

			(*close will be requested in step FRM_RBUF*)

		FRM_OPEN:	(*--- open serial interface*)

			(*Parameters for FRM_xopen()*)
			Receiver.FRM_xopen_0.enable := TRUE;
			Receiver.FRM_xopen_0.device := ADR('IF6.ST1.IF4');							(*Devicename --> see your serial interface properties*)
			Receiver.FRM_xopen_0.mode := ADR('/PHY=RS232 /BD=115200 /DB=8 /PA=E /SB=1'); (*Modestring --> specifies the seria operation mode*)
			Receiver.FRM_xopen_0.config := ADR(Receiver.xopenConfig) ;					(*Additional Parameters, optional*)

			(*Additional Parameters for FRM_xopen()*)
			Receiver.xopenConfig.idle     := 10;								(*Idle time between two characters*)
			Receiver.xopenConfig.delimc   := 0;									(*activate two delimeters*)
			Receiver.xopenConfig.delim[0] := 0; 								(*e.g. CR - carridge return -> dec 13*)
			Receiver.xopenConfig.delim[1] := 0; 								(*e.g. LF - line feed -> dec 10*)
			Receiver.xopenConfig.tx_cnt   := 3;									(*number of transmit buffers*)
			Receiver.xopenConfig.rx_cnt   := 3; 								(*number of receive buffers*)
			Receiver.xopenConfig.tx_len   := 0; 								(*length of transmit buffers*)
			Receiver.xopenConfig.rx_len   := 44; 								(*lenght of receive buffers*)
			Receiver.xopenConfig.argc     := 0;									(*activate additional options*)
			Receiver.xopenConfig.argv     := 0;									(*parameters for additional options (check help)*)

			Receiver.FRM_xopen_0();												(*call the FRM_xopen() function*)

			IF Receiver.FRM_xopen_0.status = 0 THEN
				Receiver.step := FRM_READ;										(*Interface opend successfully --> next step*)
			ELSIF Receiver.FRM_xopen_0.status = BUSY THEN
				Receiver.step := FRM_OPEN;										(*operation not finished yet --> call again*)
			ELSE
				Receiver.step := FRM_ERROR;										(*function returned errorcode --> check help*)
			END_IF

		FRM_READ:	(*--- read data from serial interface*)
			Receiver.FRM_read_0.enable := TRUE;
			Receiver.FRM_read_0.ident := Receiver.FRM_xopen_0.ident;

			Receiver.FRM_read_0();												(*call the FRM_read() function*)

			IF Receiver.FRM_read_0.status = 0 THEN
				Receiver.step := FRM_COPY_RD_DATA;								(*system returned a valid data --> next step*)
			ELSIF Receiver.FRM_read_0.status = frmERR_NOINPUT THEN
				Receiver.step := FRM_READ;										(*no data available --> call again*)
			ELSIF Receiver.FRM_read_0.status = frmERR_INPUTERROR THEN
				Receiver.step := FRM_RBUF;										(*received Frame with defective characters, skip data*)
			ELSE
				Receiver.step := FRM_ERROR;										(*function returned errorcode --> check help*)
			END_IF

		FRM_COPY_RD_DATA: (*--- copy data out of the receive buffer*)
			memset(ADR(Receiver.receive_data),0,SIZEOF(Receiver.receive_data));			(*clear read_data buffer*)
			memcpy(ADR(Receiver.receive_data),Receiver.FRM_read_0.buffer,Receiver.FRM_read_0.buflng);     (*copy and evaluate read data*)
			checkMessageValidity;
			IF messageOk THEN
				extractInsData;
			END_IF;
			Receiver.step := FRM_RBUF;													(*release read buffer*)

		FRM_RBUF:	(*--- release readbuffer*)

			(*Parameters for FRM_rbuf()*)
			Receiver.FRM_rbuf_0.enable := TRUE;
			Receiver.FRM_rbuf_0.ident := Receiver.FRM_xopen_0.ident;					(*ident from FRM_xopen()*)
			Receiver.FRM_rbuf_0.buffer := Receiver.FRM_read_0.buffer;					(*read buffer*)
			Receiver.FRM_rbuf_0.buflng := Receiver.FRM_read_0.buflng;					(*length of sendbuffer*)

			Receiver.FRM_rbuf_0();														(*call the FRM_rbuf() function*)

			IF Receiver.FRM_rbuf_0.status = 0 THEN
				IF Receiver.Commands.close = TRUE THEN
					Receiver.Commands.open_receive := FALSE;								(*disable command open_send*)
					Receiver.step := FRM_CLOSE;											(*request to close serial port*)
				ELSE
					Receiver.step := FRM_READ;											(*read again*)
				END_IF
			ELSIF Receiver.FRM_rbuf_0.status = BUSY THEN
				Receiver.step := FRM_RBUF;												(*operation not finished yet --> call again*)
			ELSIF Receiver.FRM_rbuf_0.status = frmERR_INVALIDBUFFER THEN
				Receiver.step := FRM_READ;												(*buffer is invalid --> read again*)
			ELSE
				Receiver.step := FRM_ERROR;												(*function returned errorcode --> check help*)
			END_IF

		FRM_CLOSE:	(*--- close the interface*)
			Receiver.FRM_close_0.enable := TRUE;
			Receiver.FRM_close_0.ident := Receiver.FRM_xopen_0.ident;					(*ident from FRM_xopen()*)

			Receiver.FRM_close_0();														(*call the FRM_close() function*)

			IF Receiver.FRM_close_0.status = 0 THEN
				Receiver.Commands.close := FALSE;										(*disable close command*)
				Receiver.step := FRM_WAIT;												(*closed interface successfully --> wait step*)
			ELSIF Receiver.FRM_close_0.status = BUSY THEN
				Receiver.step := FRM_CLOSE;												(*operation not finished yet --> call again*)
			ELSE
				Receiver.step := FRM_ERROR;												(*function returned errorcode --> check help*)
			END_IF

		FRM_ERROR:	(*--- error handling*)
		; (*not implementet yet, check help for error codes*)
	END_CASE

	// Publish data
	gINS.data.actLonVelocity_ms  := gINS.input.velX; 		// [km/h]
	gINS.data.actLatVelocity_ms  := gINS.input.velY; 		// [km/h]
	gINS.data.actLonVelocity_kmh := gINS.input.velX * 3.6; 	// [km/h]
	gINS.data.actLatVelocity_kmh := gINS.input.velY * 3.6; 	// [km/h]
	gINS.data.actLonAcceleration := gINS.input.accX;
	gINS.data.actLatAcceleration := gINS.input.accY;
	gINS.data.actYawRate 		 := gINS.input.gyroZ;

	(* Service actions *)

	// Calculate the distance traveled by the vehicle
	distanceMeasurement;
	// Estimate Range
	rangeEstimation;

END_PROGRAM

PROGRAM _EXIT
	MTFilterMovingAverage_0.Enable := FALSE;
	MTFilterMovingAverage_0();
END_PROGRAM
```

### Program Logical/Inverters/CAN/CAN/Receive

#### Receive_Bus.st
```iecst
ACTION Receive_Bus:

	bus[i].ArCanReceive_0(); // Run function block => Get next data frame
	FOR k := 0 TO 10 DO
		(* If a new message has been received *)
		IF bus[i].ArCanReceive_0.NewDataValid THEN
			// Update the number of messages received
			bus[i].receivedMessages := bus[i].receivedMessages + 1;

			(* Find which inverter the message came from *)
			IF    bus[i].ArCanReceive_0.ReceivedFrame.ID = (RX_CAN_ID_BASE + 16#083) OR bus[i].ArCanReceive_0.ReceivedFrame.ID = (RX_CAN_ID_BASE + 16#085) THEN
				inverterId := 0;
			ELSIF bus[i].ArCanReceive_0.ReceivedFrame.ID = (RX_CAN_ID_BASE + 16#084) OR bus[i].ArCanReceive_0.ReceivedFrame.ID = (RX_CAN_ID_BASE + 16#086) THEN
				inverterId := 1;
			ELSIF bus[i].ArCanReceive_0.ReceivedFrame.ID = (RX_CAN_ID_BASE + 16#087) OR bus[i].ArCanReceive_0.ReceivedFrame.ID = (RX_CAN_ID_BASE + 16#089) THEN
				inverterId := 2;
			ELSIF bus[i].ArCanReceive_0.ReceivedFrame.ID = (RX_CAN_ID_BASE + 16#088) OR bus[i].ArCanReceive_0.ReceivedFrame.ID = (RX_CAN_ID_BASE + 16#08A) THEN
				inverterId := 3;
			ELSE
				inverterId := 4;
			END_IF;

			// Decode the message
			IF  bus[i].ArCanReceive_0.ReceivedFrame.ID = (RX_CAN_ID_BASE + 16#083) OR bus[i].ArCanReceive_0.ReceivedFrame.ID = (RX_CAN_ID_BASE + 16#084) OR
				bus[i].ArCanReceive_0.ReceivedFrame.ID = (RX_CAN_ID_BASE + 16#087) OR bus[i].ArCanReceive_0.ReceivedFrame.ID = (RX_CAN_ID_BASE + 16#088) THEN

				Inv_ActualValue1;
			ELSE
				Inv_ActualValue2;
			END_IF;

			// Run disconnection detection routine
			updateDisconnectionDetection;

			// Get next data frame
			bus[i].ArCanReceive_0();
		ELSE
			EXIT;
		END_IF;

	END_FOR;

	gInverters.status.errorCanFramesLost[i] := bus[i].ArCanReceive_0.NumberOfLostFrames <> 0;

END_ACTION
```

### Program Logical/Inverters/Control/Control (IEC)

#### Variables.var
```iecst
VAR
	tempActivateOutputTorque : BOOL := FALSE;
	tempManualControl : BOOL := FALSE;
	distDelta : REAL;
	cycletime : UDINT;
	RTInfo_0 : RTInfo;
	constant : constant_typ;
	TON_history : TON;
	TON_acceleration_0to100 : TON;
	torqueSetpoint : ARRAY[0..3] OF REAL;
	enableAccelerationTimer : BOOL;
	i_powerLimit : INT;
	i : INT;
	j : INT;
	control : control_typ;
	torqueLimitNM : REAL;
	ActualSpeedRADS : REAL;
	MaxSpeedRADS : REAL;
	individualInverterTorqueEnabled : BOOL;
END_VAR
```

#### Program Logical/Inverters/Control/Control/Controllers

##### powerLimiter.st
```iecst
ACTION powerLimiterInit:
	// Initialize the controller values
	gInverters.data.powerLimitKW := 80;
	gInverters.data.powerLimitMargin := 0.9;

	//control.PL.enable 		 := gInverters.cmd.enablePowerLimiter;
	//control.PL.MAX_POWER	 := gInverters.data.powerLimitKW; // [kW]
	//FOR i := 0 TO INVERTER_COUNT DO
	//	control.PL.I_GAIN[i] := 0;
	//	control.PL.P_GAIN[i] := 0;
	//END_FOR;
	constant.NOMINAL_TORQUE := 9.8; // [Nm]
	constant.MAX_TORQUE 	:= 21; // [Nm]
END_ACTION

ACTION powerLimiterCyclic:
	// Service the controller
	gInverters.data.MaxSpeedRPM :=  MAX(gInverters.inverter[0].data.actualVelocity, gInverters.inverter[1].data.actualVelocity, gInverters.inverter[2].data.actualVelocity, gInverters.inverter[3].data.actualVelocity, 1);
	MaxSpeedRADS := (gInverters.data.MaxSpeedRPM*2*constant.PI)/60;
	torqueLimitNM := ((MIN(gInverters.data.powerLimitKW,gORION.data.DCL_KW) /4)*1000)/MaxSpeedRADS * gInverters.data.powerLimitMargin; // 0.9 is equvivalent to 10% margin of limit
	gInverters.inverter[i].outputs.com_torqueLimitPos 	:= DINT_TO_INT(LIMIT(0,REAL_TO_DINT((torqueLimitNM/constant.NOMINAL_TORQUE)*1000), 32767)); // Is sent as 0.1% of nominel torque

	//control.PL.enable 				:= gInverters.cmd.enablePowerLimiter; // This might needed to be turned on?
	//control.PL.act_power			:= gShunt.data.actPowerKW;
	//control.PL.lowest_cell_voltage 	:= MIN(gAMS.data.cellVoltageMin[0], gAMS.data.cellVoltageMin[1], gAMS.data.cellVoltageMin[2], gAMS.data.cellVoltageMin[3], gAMS.data.cellVoltageMin[4]);
	//control.PL();
END_ACTION

ACTION powerLimiterCyclicIndividual:
	// Service the controller
	ActualSpeedRADS := (MAX(gInverters.inverter[i].data.actualVelocity, 1)*2*constant.PI)/60;
	torqueLimitNM := (gInverters.data.powerLimitKwInverter[i]*1000)/ActualSpeedRADS * gInverters.data.powerLimitMargin; // 0.9 is equvivalent to 10% margin of limit
	gInverters.inverter[i].outputs.com_torqueLimitPos 	:= DINT_TO_INT(LIMIT(0,REAL_TO_DINT((torqueLimitNM/constant.NOMINAL_TORQUE)*1000), 32767)); // Is sent as 0.1% of nominel torque

	//control.PL.enable 				:= gInverters.cmd.enablePowerLimiter; // This might needed to be turned on?
	//control.PL.act_power			:= gShunt.data.actPowerKW;
	//control.PL.lowest_cell_voltage 	:= MIN(gAMS.data.cellVoltageMin[0], gAMS.data.cellVoltageMin[1], gAMS.data.cellVoltageMin[2], gAMS.data.cellVoltageMin[3], gAMS.data.cellVoltageMin[4]);
	//control.PL();
END_ACTION
```

#### torqueOff.st
```iecst
(* Test if both brake and torque pedal is pressed at the same time. If so turn on torque until both pedals has been released again *)
ACTION torqueOff:
	// If inverter are allowed to shut eachother down parse through each pair and check if it should shut its partner down
	IF gInverters.cmd.enableMotorPairShutdown THEN
		(* Front *)
		gInverters.inverter[1].cmd.shutdownByPartner := gInverters.inverter[0].status.errorTimeout;
		gInverters.inverter[0].cmd.shutdownByPartner := gInverters.inverter[1].status.errorTimeout;

		(* Rear *)
		gInverters.inverter[3].cmd.shutdownByPartner := gInverters.inverter[2].status.errorTimeout;
		gInverters.inverter[2].cmd.shutdownByPartner := gInverters.inverter[3].status.errorTimeout;
	ELSE
		// Else let all inverters run for themselves
		FOR i := 0 TO INVERTER_COUNT DO
			gInverters.inverter[i].cmd.shutdownByPartner := FALSE;
		END_FOR;
	END_IF;

	(* Output actual torque *)
	FOR i := 0 TO INVERTER_COUNT DO
		gInverters.inverter[i].outputs.torqueEnable := gTorqueSensor.status.torqueEnabled AND NOT (gInverters.inverter[i].cmd.shutdownByPartner OR gInverters.inverter[i].status.errorTimeout);
	END_FOR;
	IF NOT gInverters.cmd.manualControl THEN
		IF gInverters.cmd.enableMotorPairShutdown THEN
			gInverters.output.do_enableInv12 := gInverters.inverter[0].outputs.torqueEnable AND gInverters.inverter[1].outputs.torqueEnable;
			gInverters.output.do_enableInv34 := gInverters.inverter[2].outputs.torqueEnable AND gInverters.inverter[3].outputs.torqueEnable;
		END_IF;
	END_IF;

END_ACTION
```

### Program Logical/Inverters/Inv_statemachine/Inv_statemachine (IEC)

#### mission.st
```iecst
ACTION missionInit:

	missions.missionList[MISSION_NONE] 			:= 'Mission None';
	missions.missionList[MISSION_ACCELERATION] 	:= 'Mission Acceleration';
	missions.missionList[MISSION_SKIDPAD] 		:= 'Mission Skidpad';
	missions.missionList[MISSION_SPRINT] 		:= 'Mission Sprint';
	missions.missionList[MISSION_ENDURANCE] 	:= 'Mission Endurance';
	missions.missionList[MISSION_BRAKE_TEST] 	:= 'Mission Brake Test';
	missions.missionList[MISSION_TESTING] 		:= 'Mission Testing';

	gStateMachine.status.missionIndex 		:= MISSION_NONE;

	IF gIsSimulation THEN
		missions.MpRecipeXml_0.DeviceName 	:= ADR('C');
	ELSE
		missions.MpRecipeXml_0.DeviceName 	:= ADR('plc');
	END_IF;
	missions.MpRecipeXml_0.FileName 	:= ADR('mission_none');
	missions.MpRecipeXml_0.MpLink 		:= ADR(gRecipeXml);
	missions.MpRecipeXml_0.Enable 		:= TRUE;

	missions.MpRecipeRegPar_0[0].PVName := ADR('gInverters.data.powerLimitKW');
	missions.MpRecipeRegPar_0[1].PVName := ADR('gInverters.data.torqueLimitNm');
	missions.MpRecipeRegPar_0[2].PVName := ADR('gInverters.cmd.enableLaunchProfile');
	missions.MpRecipeRegPar_0[3].PVName := ADR('gInverters.cmd.enablePowerLimiter');
	missions.MpRecipeRegPar_0[4].PVName := ADR('gInverters.cmd.enableRegenerativeBraking');
	missions.MpRecipeRegPar_0[5].PVName := ADR('gInverters.cmd.enableTorqueVectoring');
	missions.MpRecipeRegPar_0[6].PVName := ADR('gInverters.cmd.enableTractionControl');
	missions.MpRecipeRegPar_0[7].PVName := ADR('gInverters.cmd.enableMotorPairShutdown');
	missions.MpRecipeRegPar_0[8].PVName := ADR('gInverters.cmd.enableConfigurationDuringDrive');
	missions.MpRecipeRegPar_0[9].PVName := ADR('gInverters.status.deratingStaticPercent');

	FOR i := 0 TO MAX_MISSION_PARAMETERS DO
		missions.MpRecipeRegPar_0[i].Enable := TRUE;
		missions.MpRecipeRegPar_0[i].MpLink := ADR(gRecipeXml);
	END_FOR;

	// Initialize to TRUE so the car will start by fetching the current mission data
	gStateMachine.cmd.changeMission 	:= TRUE;

END_ACTION

ACTION missionCyclic:
	gStateMachine.status.mission := missions.missionList[gStateMachine.status.missionIndex];

	(* detect a mission change *)
	IF gStateMachine.status.missionIndex <> missions.missionOld THEN
		gStateMachine.cmd.changeMission := TRUE;
		missions.missionOld 			:= gStateMachine.status.missionIndex;
	END_IF;

	(* If the mission has been change load the mission config *)
	IF (gStateMachine.cmd.changeMission OR gStateMachine.cmd.loadMission) AND gInverters.status.configurationEnabled THEN
		gStateMachine.cmd.changeMission := FALSE;
		gStateMachine.cmd.loadMission := FALSE;
//		gDashboard.cmd.sendVehicleConfigMsg := TRUE; // Transmit new mission to dashboard
//		CASE gStateMachine.status.missionIndex OF
//			MISSION_NONE: 		  missions.MpRecipeXml_0(FileName := ADR('mission_none'		 	));
//			MISSION_ACCELERATION: missions.MpRecipeXml_0(FileName := ADR('mission_acceleration'	));
//			MISSION_SKIDPAD: 	  missions.MpRecipeXml_0(FileName := ADR('mission_skidpad'	 	));
//			MISSION_SPRINT: 	  missions.MpRecipeXml_0(FileName := ADR('mission_sprint'		));
//			MISSION_ENDURANCE: 	  missions.MpRecipeXml_0(FileName := ADR('mission_endurance'	));
//			MISSION_BRAKE_TEST:   missions.MpRecipeXml_0(FileName := ADR('mission_brake_test'	));
//			MISSION_TESTING: 	  missions.MpRecipeXml_0(FileName := ADR('mission_testing'	 	));
//		END_CASE
		missions.MpRecipeXml_0(Load := TRUE);
	END_IF;

	(* Save current configuration to current mission *)
	IF gStateMachine.cmd.saveMission THEN
		gStateMachine.cmd.saveMission := FALSE;
		missions.MpRecipeXml_0(Save := TRUE);
	END_IF;

	(* Run function blocks *)
	FOR i := 0 TO MAX_MISSION_PARAMETERS DO
		missions.MpRecipeRegPar_0[i]();
	END_FOR;
	missions.MpRecipeXml_0(Save := FALSE, Load := FALSE);

END_ACTION
```

### Library Logical/Libraries/brdkSIM (ANSIC)
Depends on: AsIO, AsBrStr, sys_lib

#### brdkSIM.fun - Exported functions and function blocks
```iecst
FUNCTION_BLOCK brdkSimInput (*TODO: Add your comment here*) (*$GROUP=User,$CAT=User,$GROUPICON=User.png,$CATICON=User.png*)
	VAR_INPUT
		enable : BOOL;
		dpName : STRING[100];
		setValue : UDINT;
	END_VAR
	VAR_OUTPUT
		status : brdkSIM_status_typ;
	END_VAR
	VAR
		internal : brdkSimInput_internal_typ;
	END_VAR
END_FUNCTION_BLOCK

FUNCTION_BLOCK brdkSimOutput (*TODO: Add your comment here*) (*$GROUP=User,$CAT=User,$GROUPICON=User.png,$CATICON=User.png*)
	VAR_INPUT
		enable : BOOL;
		pvName : STRING[100];
	END_VAR
	VAR_OUTPUT
		actValue : UDINT;
		status : brdkSIM_status_typ;
	END_VAR
	VAR
		internal : brdkSimOutput_internal_typ;
	END_VAR
END_FUNCTION_BLOCK
```

- Library Logical/Libraries/brdkSTR (ANSIC, version 1.03.1) (no source held here)

### brdkUSB.typ
```iecst
TYPE
	brdk_usb_status_typ :
		( (*Status of the function block*)
		BRDK_USB_STATUS_NO_USB_DEV_FOUND := 0, (*No USB device found*)
		BRDK_USB_STATUS_FB_READY := 1 (*Ready to connect*)
		);
	brdk_usb_connect_node_output_typ : 	STRUCT  (*Node device info*)
		device : STRING[5]; (*Node device name*)
		freeMemory : DINT; (*[Mb] -1 means memory info could not be read*)
		totalMemory : DINT; (*[Mb] -1 means memory info could not be read*)
	END_STRUCT;
	brdk_usb_connect_internal_typ : 	STRUCT  (*internal variables*)
		UsbNodeListGet_0 : UsbNodeListGet; (*get node list*)
		nodeIdBuffer : ARRAY[0..BRDK_USB_MAX_DEVICES]OF UDINT; (*node id buffer*)
		oldCnt : UDINT; (*old count*)
		node : ARRAY[0..BRDK_USB_MAX_DEVICES]OF brdk_usb_connect_int_node_typ; (*node list*)
		simulationMountActivated : BOOL; (*is the mount being simulated*)
	END_STRUCT;
	brdk_usb_connect_int_node_typ : 	STRUCT  (*internal node variables*)
		state : UINT; (*node state*)
		infoBuffer : usbNode_typ; (*node info*)
		UsbNodeGet_0 : UsbNodeGet; (*usb get node*)
		DevLink_0 : DevLink; (*creates a deveice link*)
		DevUnlink_0 : DevUnlink; (*unlinks a device link*)
		DevMemInfo_0 : DevMemInfo; (*reads the memory info about the device*)
		device : STRING[8]; (*device name*)
		param : STRING[20]; (*device parameters*)
		devLinkFailCnt : UDINT; (*faild dev link count*)
	END_STRUCT;
END_TYPE
```

### Library Logical/Libraries/sduVikings (IEC)

#### sduVikings.fun - Exported functions and function blocks
```iecst
{REDUND_ERROR} FUNCTION_BLOCK calculateSensorNetOut (*TODO: Add your comment here*) (*$GROUP=User,$CAT=User,$GROUPICON=User.png,$CATICON=User.png*)
	VAR_INPUT
		input : {REDUND_UNREPLICABLE} INT;
		polyCoeffs : {REDUND_UNREPLICABLE} ARRAY[0..8] OF REAL;
	END_VAR
	VAR_OUTPUT
		output : {REDUND_UNREPLICABLE} REAL;
	END_VAR
	VAR
		i : USINT;
		y : REAL;
	END_VAR
END_FUNCTION_BLOCK

FUNCTION_BLOCK torqueVectoring
	VAR_INPUT
		enable : BOOL;
		torque_input : REAL;
		steering_angle : REAL;
		MAX_DERATING : REAL;
		MAX_STEERING_ANGLE : REAL;
	END_VAR
	VAR_OUTPUT
		torque_output : ARRAY[0..3] OF REAL;
	END_VAR
	VAR
		i : USINT;
	END_VAR
END_FUNCTION_BLOCK

FUNCTION_BLOCK tractionControl
	VAR_INPUT
		enable : BOOL;
		longitudinal_wheel_slip : ARRAY[0..3] OF REAL;
		LON_SLIP_REF : REAL;
		P_GAIN : ARRAY[0..3] OF REAL;
		I_GAIN : ARRAY[0..3] OF REAL;
	END_VAR
	VAR_OUTPUT
		derating_output : ARRAY[0..3] OF REAL;
	END_VAR
	VAR
		i : USINT;
	END_VAR
END_FUNCTION_BLOCK

FUNCTION_BLOCK powerLimiter
	VAR_INPUT
		enable : BOOL;
		act_power : REAL;
		lowest_cell_voltage : REAL;
		MAX_POWER : REAL;
		P_GAIN : ARRAY[0..3] OF REAL;
		I_GAIN : ARRAY[0..3] OF REAL;
	END_VAR
	VAR_OUTPUT
		derating_output : ARRAY[0..3] OF REAL;
	END_VAR
	VAR
		i : USINT;
	END_VAR
END_FUNCTION_BLOCK

FUNCTION_BLOCK launchProfile
	VAR_INPUT
		enable : BOOL;
		act_lon_velocity : REAL;
	END_VAR
	VAR_OUTPUT
		derating_output : ARRAY[0..3] OF REAL;
	END_VAR
	VAR
		i : USINT;
	END_VAR
END_FUNCTION_BLOCK

FUNCTION_BLOCK torqueLimiter
	VAR_INPUT
		enable : BOOL;
		max_torque : REAL;
	END_VAR
	VAR_OUTPUT
		derating_output : ARRAY[0..3] OF REAL;
	END_VAR
	VAR
		i : USINT;
	END_VAR
END_FUNCTION_BLOCK

{REDUND_ERROR} FUNCTION_BLOCK regenerativeBraking (*TODO: Add your comment here*) (*$GROUP=User,$CAT=User,$GROUPICON=User.png,$CATICON=User.png*)
	VAR_INPUT
		enable : BOOL;
		vehicle_lon_velocity : REAL;
		negative_torque_transfer : REAL;
		torque_pedal : REAL;
		brake_pressure : REAL;
		REGEN_BRAKING_GAIN : REAL;
		IDLE_MOTOR_TORQUE : REAL;
	END_VAR
	VAR_OUTPUT
		negative_torque_limit : ARRAY[0..3] OF REAL;
		positive_torque_limit : ARRAY[0..3] OF REAL;
	END_VAR
	VAR
		negTrqLimSetpoint : ARRAY[0..3] OF REAL;
		i : USINT;
	END_VAR
END_FUNCTION_BLOCK
```

#### torqueVectoring.st
```iecst
FUNCTION_BLOCK torqueVectoring

	IF enable THEN

	ELSE
		// If TV is disabled. Parse torque pedal signal through
		FOR i := 0 TO 3 DO
			torque_output[i] := torque_input;
		END_FOR;
	END_IF;

END_FUNCTION_BLOCK
```

#### powerLimiter.st
```iecst
FUNCTION_BLOCK powerLimiter
	IF enable THEN

	ELSE
		FOR i := 0 TO 3 DO
			derating_output[i] := 1;
		END_FOR;
	END_IF;

END_FUNCTION_BLOCK
```

### Program Logical/Libraries/VhclDyn/TorqueLimiting

#### TL_SetTorqueLimit.st
```iecst
(* TODO: Add your comment here *)
FUNCTION_BLOCK TL_SetTorqueLimit
	output := LIMIT(0,torqueLimit/100.00,1);
END_FUNCTION_BLOCK
```

### Program Logical/Misc/AlarmManagement/AlarmManagement

#### Variables.var
```iecst
VAR
	MpAlarmXListUI_0 : MpAlarmXListUI;
	MpAlarmXListUIConnectType_0 : MpAlarmXListUIConnectType;
	MpAlarmXCore_0 : MpAlarmXCore;
END_VAR
```

#### Main.st
```iecst
PROGRAM _INIT
	MpAlarmXCore_0.MpLink 		:= ADR(gAlarmXCore);
	MpAlarmXCore_0.Enable 		:= TRUE;

	MpAlarmXListUI_0.MpLink 	:= ADR(gAlarmXCore);
	MpAlarmXListUI_0.UIConnect 	:= ADR(MpAlarmXListUIConnectType_0);
	MpAlarmXListUI_0.Enable 	:= TRUE;

END_PROGRAM

PROGRAM _CYCLIC
	(* Alarm *)
	MpAlarmXCore_0();
	MpAlarmXListUI_0();

END_PROGRAM

PROGRAM _EXIT

	MpAlarmXCore_0(Enable:=FALSE);
	MpAlarmXListUI_0(Enable:=FALSE);

END_PROGRAM
```

### Program Logical/Misc/DataLogging/sampleST (IEC)

#### Variables.var
```iecst
VAR
	i : USINT;
	this : brdkusb_sample_st_interal_typ;
END_VAR
```

### Program Logical/Misc/DataLogging/DataLog (IEC)

#### initSetup.st
```iecst
	//(* Writing the data to be datalogged *)
ACTION initSetup:
	// State
	gDataLogging.data.csvData[0] := 'gStateMachine.status.stateName';
	// Mission
	gDataLogging.data.csvData[1] := 'gStateMachine.status.mission';
	// Instruction
	gDataLogging.data.csvData[2] := 'gStateMachine.status.instruction';

	// ******* Dashboard information
	// State
	gDataLogging.data.csvData[3] := 'gDashboard.status.DashboardDisconnected';
	gDataLogging.data.csvData[4] := 'gDashboard.status.errorCode';
	// Buttons
	gDataLogging.data.csvData[5] := 'gDashboard.inputs.di_button1';
	gDataLogging.data.csvData[6] := 'gDashboard.inputs.di_button2';
	gDataLogging.data.csvData[7] := 'gDashboard.inputs.di_button3';
	gDataLogging.data.csvData[8] := 'gDashboard.inputs.di_button4';
	gDataLogging.data.csvData[9] := 'gDashboard.inputs.di_buttonSafety';
	gDataLogging.data.csvData[10] := 'gDashboard.inputs.di_buttonTractive';
	gDataLogging.data.csvData[11] := 'gDashboard.inputs.di_buttonDrive';

	// LED's
	gDataLogging.data.csvData[12] := 'gDashboard.outputs.do_ledAMS';
	gDataLogging.data.csvData[13] := 'gDashboard.outputs.do_ledIMD';
	gDataLogging.data.csvData[14] := 'gDashboard.outputs.do_ledLV';
	gDataLogging.data.csvData[15] := 'gDashboard.outputs.do_ledREADY';
	gDataLogging.data.csvData[16] := 'gDashboard.outputs.do_ledSC';
	gDataLogging.data.csvData[17] := 'gDashboard.outputs.do_ledTS_OFF';

END_ACTION
```

### globalDataLogging.typ
```iecst
TYPE
	gDataLogging_typ : 	STRUCT
		status : gDataLogging_status_typ;
		inputs : gDataLogging_inputs_typ;
		outputs : gDataLogging_outputs_typ;
		data : gDataLogging_data_typ;
	END_STRUCT;
	gDataLogging_status_typ : 	STRUCT
		dataloggingActive : BOOL;
	END_STRUCT;
	gDataLogging_inputs_typ : 	STRUCT
		dummy : UINT;
	END_STRUCT;
	gDataLogging_outputs_typ : 	STRUCT
		dummy : BOOL;
	END_STRUCT;
	gDataLogging_data_typ : 	STRUCT
		csvData : ARRAY[0..DATALOG_MAX_LOG_VARS]OF STRING[80];
	END_STRUCT;
END_TYPE
```

### globalSafetyChain.var
```iecst
VAR
	gSafetyChain : gSafetyChain_typ;
END_VAR
VAR CONSTANT
	MAX_SC_ELEMENTS : USINT := 26;
END_VAR
```

### Program Logical/SC/SafetyChain (IEC)

#### Main.st - Init, cyclic, exit code
```iecst
PROGRAM _INIT

	(* Write the sc error names into an array *)
	scStrings;

	gSafetyChain.inputs.di_LVMS_OK := TRUE;

END_PROGRAM

PROGRAM _CYCLIC

	// Read data into SC
	gSafetyChain.inputs.interlockHVDC_OK 	:= NOT gAMS.status.error.hvdcInterlockError; // Might be NOT, depends on how the signal from the CAN is
	gSafetyChain.inputs.IMD_OK 				:= gSafetyChain.inputs.interlockHVDC_OK AND NOT gAMS.status.error.imdError;
	gSafetyChain.inputs.AMS_OK 				:= gSafetyChain.inputs.interlockHVDC_OK AND NOT gAMS.status.error.amsError;

	(* Write all safety chain elements into an array ready for parsing through *)
	scUpdate;

	(* Go through all safety chain elements and check if they are broken or not *)
	FOR i := 0 TO MAX_SC_ELEMENTS DO
		IF NOT gSafetyChain.status.sc[i] THEN
			gSafetyChain.status.scErrorString 	:= gSafetyChain.status.scErrorStrings[i];
			gSafetyChain.status.scErrorIndex 	:= i;
			EXIT;
		END_IF
	END_FOR

	(* check all parts of the safety chain *)
//	gSafetyChain.status.scOK_notEnabled := gSafetyChain.inputs.di_TSMS_OK;

	gSafetyChain.status.scOK_notEnabled := 		gSafetyChain.inputs.AMS_OK
											AND gSafetyChain.inputs.di_BOTS_OK
											AND gSafetyChain.inputs.di_TS_Container
											AND gSafetyChain.inputs.di_BSPD_OK
											AND gSafetyChain.inputs.di_interlockHVD_OK
											AND gSafetyChain.inputs.IMD_OK
											AND gSafetyChain.inputs.di_inertiaSwitch_OK
											AND gSafetyChain.inputs.di_interlockMotorFL_OK
											AND gSafetyChain.inputs.di_interlockMotorFR_OK
											AND gSafetyChain.inputs.di_interlockMotorRL_OK
											AND gSafetyChain.inputs.di_interlockMotorRR_OK
											AND gSafetyChain.inputs.di_interlockTSMP_OK
											AND gSafetyChain.inputs.di_interlockWheelFL_OK
											AND gSafetyChain.inputs.di_interlockWheelFR_OK
											AND gSafetyChain.inputs.di_interlockWheelRL_OK
											AND gSafetyChain.inputs.di_interlockWheelRR_OK
											AND gSafetyChain.inputs.interlockHVDC_OK
											AND gSafetyChain.inputs.di_LVMS_OK
											AND gSafetyChain.inputs.di_supply
											AND gSafetyChain.inputs.di_shutdownCockpit_OK
											AND gSafetyChain.inputs.di_shutdownLeft_OK
											AND gSafetyChain.inputs.di_shutdownRight_OK
											AND gSafetyChain.inputs.di_TSMS_OK;

	(* Get the safety chain status including the enable switch *)
	gSafetyChain.status.scOK := 	gSafetyChain.status.scOK_notEnabled AND gAMS.status.scEnabled;

	// Make a version of the scOK signal that is more robust towards noise and flicker on the shutdown circuit lines
	IF gStateMachine.status.state = STATE_ENABLING_SC OR gStateMachine.status.state = STATE_PRECHARGING THEN
		// When waiting for the AMS the SC experiences many spikes and the delay is therefore made very big to not falsely trigger.
		TON_persistancetimer.PT := T#10000ms;
	ELSE
		// Under normal conditions the SC should be concluded broken after 1 sec.
		TON_persistancetimer.PT := T#1000ms;
	END_IF;

	TON_persistancetimer.IN := NOT gSafetyChain.status.scOK;
	TON_persistancetimer();

	gSafetyChain.status.scOKPersistent := NOT TON_persistancetimer.Q;

	IF EDGENEG(gSafetyChain.status.scOKPersistent) THEN
		gEventLog.newEventString := 'SC Broken at: ';
		strcat(ADR(gEventLog.newEventString), ADR(gSafetyChain.status.scErrorString));
		logEvent;
	END_IF;

	(* Convert the SC status to USINT. This is used for the liveview to select a picture displaying the status *)
	IF gSafetyChain.status.scOK_notEnabled THEN
		gSafetyChain.status.scOK_usint := 1;
	ELSIF gSafetyChain.status.scOKPersistent THEN
		gSafetyChain.status.scOK_usint := 2;
	ELSE
		gSafetyChain.status.scOK_usint := 0;
	END_IF

END_PROGRAM

PROGRAM _EXIT

END_PROGRAM
```

### Program Logical/SensorNet/globalSensorNet (IEC)

#### Variables.var
```iecst
VAR
	a : ARRAY[0..SENSOR_NET_POLY_LEN] OF REAL;
	i : USINT;
	y : REAL;
	x : INT;
	calculateSensorNetOut_0 : calculateSensorNetOut;
END_VAR
```

### globalSteeringAngle.typ
```iecst
TYPE
	gSteeringAngle_cmd_typ : 	STRUCT
		angleSensor : INT;
	END_STRUCT;
	gSteeringAngle_typ : 	STRUCT
		status : gSteeringAngle_status_typ;
		inputs : gSteeringAngle_inputs_typ;
		outputs : gSteeringAngle_outputs_typ;
		data : gSteeringAngle_data_typ;
		cmd : gSteeringAngle_cmd_typ;
	END_STRUCT;
	gSteeringAngle_status_typ : 	STRUCT
		ok : BOOL;
		error : BOOL;
		errorOutOfRange : BOOL;
		disconnected : BOOL;
		steeringWheelSVG : STRING[1000];
		wheelSVG : STRING[300];
	END_STRUCT;
	gSteeringAngle_data_typ : 	STRUCT
		angleDegrees : REAL;
		wheelAngle : REAL;
	END_STRUCT;
	gSteeringAngle_inputs_typ : 	STRUCT
		angleSensor : INT;
	END_STRUCT;
	gSteeringAngle_outputs_typ : 	STRUCT
		dummy : USINT;
	END_STRUCT;
END_TYPE
```

### globalSteeringAngle.var
```iecst
VAR
	gSteeringAngle : gSteeringAngle_typ;
END_VAR
```

### Program Logical/Sensors/Sensors

#### Variables.var
```iecst
VAR
	brakingPedalVariables : braking_pedal_variables_typ;
	brakingPedalConstants : braking_pedal_constants_typ;
	torquePedalConstants : torque_pedal_constants_typ;
	torquePedalVariables : torque_pedal_variables_typ;
	steeringAngleConstants : steering_angle_constants_typ;
	steeringAngleVariables : steering_angle_variables_typ;
	lvBatteryConstants : lv_battery_constants_typ;
	lvBatteryVariables : lv_battery_variable_typ;
END_VAR
VAR RETAIN
	maxTorquePercentThrottle : USINT;
END_VAR
```

#### Main.st
```iecst
PROGRAM _INIT
	(* Initialize all the sensors *)
	// Braking Pedal Sensor
	BrakingPedalInit;

	// Torque Pedal Sensor
	TorquePedalInit;

	// Steering Angle Sensor
	SteeringAngleInit;

	// Low voltage battery
	LowVoltageBatteryInit;
END_PROGRAM

PROGRAM _CYCLIC

	// Handle Braking Pedal Sensor
	BrakingPedal;

	// Handle TorquePedal Sensor
	TorquePedal;

	// Handle Braking Pedal Sensor
	SteeringAngle;

	// Low voltage battery
	LowVoltageBattery;
END_PROGRAM

PROGRAM _EXIT
	(* Insert code here *)

END_PROGRAM
```

#### Program Logical/Sensors/Sensors/SteeringAngle

##### SteeringAngle.st
```iecst
ACTION SteeringAngleInit:
	(* Sensor limit values *)
	steeringAngleVariables.leftValue 	:= 1000;
	steeringAngleVariables.rightValue 	:= 10000;

	(* Error detection values *)
	steeringAngleConstants.disconnectionLimit := 300;
	steeringAngleConstants.lowLimit 	:= steeringAngleVariables.leftValue  - 500;
	steeringAngleConstants.highLimit 	:= steeringAngleVariables.rightValue + 500;

	steeringAngleConstants.MAX_ANGLE 	:=  100.00;
	steeringAngleConstants.MIN_ANGLE 	:= -100.00;
END_ACTION

ACTION SteeringAngle:
	(* 	Check if sensor input is within working range
		If not report an error  	*)
	gSteeringAngle.status.disconnected := INT_TO_UINT(gSteeringAngle.inputs.angleSensor) < steeringAngleConstants.disconnectionLimit;
	gSteeringAngle.status.errorOutOfRange := (NOT gSteeringAngle.status.disconnected) AND (INT_TO_UINT(gSteeringAngle.inputs.angleSensor) > steeringAngleConstants.highLimit OR INT_TO_UINT(gSteeringAngle.inputs.angleSensor) < steeringAngleConstants.lowLimit);
	(* Summerize errors *)
	gSteeringAngle.status.error := gSteeringAngle.status.disconnected OR gSteeringAngle.status.errorOutOfRange;

	(* Calculate steering angle *)
	IF NOT gSteeringAngle.status.error THEN
		// No error
		IF INT_TO_UINT(gSteeringAngle.inputs.angleSensor) < steeringAngleVariables.leftValue THEN
			gSteeringAngle.data.angleDegrees := steeringAngleConstants.MIN_ANGLE;
		ELSIF INT_TO_UINT(gSteeringAngle.inputs.angleSensor) > steeringAngleVariables.rightValue THEN
			gSteeringAngle.data.angleDegrees := steeringAngleConstants.MAX_ANGLE;
		ELSE
			gSteeringAngle.data.angleDegrees := LIMIT(-100, (INT_TO_REAL(gSteeringAngle.inputs.angleSensor) - UINT_TO_REAL(steeringAngleVariables.leftValue))/(UINT_TO_REAL(steeringAngleVariables.rightValue) - UINT_TO_REAL(steeringAngleVariables.leftValue)) *
			(ABS(steeringAngleConstants.MAX_ANGLE) + ABS(steeringAngleConstants.MIN_ANGLE)) + steeringAngleConstants.MIN_ANGLE, 100);
		END_IF;
	ELSE
		// Error
		gSteeringAngle.data.angleDegrees := 0;
	END_IF

	(* Determine if the steering angle sensor is working properly *)
	gSteeringAngle.status.ok := NOT gSteeringAngle.status.disconnected AND NOT gSteeringAngle.status.error;

	// Visualization action
	hmi;

END_ACTION
```

### Variables.var
```iecst
VAR
	TON_stateTimeout : TON;
	brdkSimInput_0 : ARRAY[0..SIM_INPUTS] OF brdkSimInput;
	this : this_typ;
END_VAR
VAR CONSTANT
	SIM_INPUTS : USINT := 50;
END_VAR
VAR
	i : USINT;
	TON_stateChange : TON;
END_VAR
```

### Program Logical/SM/StateMachine/functions

#### instruction.st
```iecst
ACTION initInstructions:
	this.instructionList[INST_INITIALIZING] 			:= 'Initializing';
	this.instructionList[INST_PRESS_SAFETY_BUTTON] 		:= 'Press Safety Button';
	this.instructionList[INST_SC_NOT_ENABLED]			:= 'Wait for SC to be Enabled';
	this.instructionList[INST_PRESS_TRACTIVE_BUTTON] 	:= 'Press Tractive Button';
	this.instructionList[INST_AMS_NOT_READY]			:= 'Wait for AMS to be Ready';
	this.instructionList[INST_PRESS_BRAKE] 				:= 'Press Brake Predal';
	this.instructionList[INST_TORQUE_PEDAL_FAULT] 		:= 'Torque Pedal Fault';
	this.instructionList[INST_PRE_CHARGING] 			:= 'Pre-Charging. Wait';
	this.instructionList[INST_PRESS_DRIVE_BUTTON] 		:= 'Press Drive Button';
	this.instructionList[INST_FIX_ERROR] 				:= 'Remove Error';
	this.instructionList[INST_CLOSE_SAFETY_CHAIN] 		:= 'Close Shutdown Circuit';
	this.instructionList[INST_IN_DRIVE] 				:= 'To Exit Drive: Press Shutdown Button';
END_ACTION

ACTION instruction:
	gStateMachine.status.instruction := this.instructionList[gStateMachine.status.instructionIndex];
END_ACTION
```

### Program Logical/SM/StateMachine/states

#### stateDrive.st
```iecst
(* State Drive *)
ACTION stateDrive:
	(* Update instruction string *)
	gStateMachine.status.instructionIndex 	:= INST_IN_DRIVE;
END_ACTION

(* Conditions for state change for STATE_DRIVE *)
ACTION stateChangeDrive:
	IF gStateMachine.status.stateChangeAllowed THEN

		(* If safety chain is broken go to state 'stateError' *)
		IF NOT gSafetyChain.status.scOKPersistent THEN
			gStateMachine.status.state 	:= STATE_ERROR;
			gAMS.cmd.abort 				:= TRUE;
		END_IF

		(* If torque pedals get too far away from eachother. Exit drive and go to tractive *)
		IF gTorqueSensor.status.plausibilityError OR gInverters.cmd.exitDrive THEN
			gStateMachine.status.state := STATE_TRACTIVE;
		END_IF
	END_IF;

END_ACTION
```

#### stateError.st
```iecst
(* State State Error *)
ACTION stateError:
	// gAMS.cmd.abort := TRUE;

END_ACTION

(* Conditions for state change for STATE_ERROR *)
ACTION stateChangeError:
	IF gStateMachine.status.stateChangeAllowed THEN
		(* Update instruction string *)
		IF NOT gSafetyChain.status.scOK_notEnabled THEN
			// Safety chain is not alright
			gStateMachine.status.instructionIndex := INST_CLOSE_SAFETY_CHAIN;
		ELSE
			// Safety chain is alright. Some other problem is active
			gStateMachine.status.instructionIndex := INST_FIX_ERROR;
		END_IF;

		(* If safety chain is OK *)
		IF gSafetyChain.status.scOK_notEnabled AND NOT gTorqueSensor.status.criticalError THEN
			gAMS.cmd.abort := FALSE;
			gStateMachine.status.state := STATE_IDLE;
		END_IF
	END_IF;

END_ACTION
```

#### stateIdle.st
```iecst
(* State Ready *)
ACTION stateIdle:

END_ACTION

(* Conditions for state change for STATE_READY *)
ACTION stateChangeIdle:
	IF gStateMachine.status.stateChangeAllowed THEN

		(* Update instruction string *)
		gStateMachine.status.instructionIndex := INST_PRESS_SAFETY_BUTTON;

		(* If safety button is pressed enable safety chain *)
		IF EDGEPOS(gDashboard.inputs.di_buttonSafety) THEN
			gStateMachine.status.state 	:= STATE_ENABLING_SC;
			gAMS.cmd.enableSC 			:= TRUE;

			(* If the PLC is simulated reset the button *)
			IF gIsSimulation THEN
				gDashboard.inputs.di_buttonSafety := FALSE;
			END_IF
		END_IF

		(* If safety chain is broken go to state 'stateError' *)
		IF NOT gSafetyChain.status.scOK_notEnabled THEN
			gStateMachine.status.state 	:= STATE_ERROR;
			gAMS.cmd.abort 				:= TRUE;
		END_IF
	END_IF;
END_ACTION
```

#### stateSCEnabled.st
```iecst
(* State Safety Chain Enabled *)
ACTION stateSCEnabled:

END_ACTION

(* Conditions for state change for STATE_SAFETY_CHAIN_ENABLED *)
ACTION stateChangeSCEnabled:
	IF gStateMachine.status.stateChangeAllowed THEN

		(* Update instruction string *)
		gStateMachine.status.instructionIndex := INST_PRESS_TRACTIVE_BUTTON;

		(* If tractive button pressed change state to 'stateOpeningRelays' *)
		IF EDGEPOS(gDashboard.inputs.di_buttonTractive) THEN
			gStateMachine.status.state 	:= STATE_PRECHARGING;
			gAMS.cmd.startPrecharge 	:= TRUE;

			(* If the PLC is simulated reset the button *)
			IF gIsSimulation THEN
				gDashboard.inputs.di_buttonTractive := FALSE;
			END_IF
		END_IF

		(* If safety chain is broken go to state 'stateError' *)
		IF NOT gSafetyChain.status.scOKPersistent THEN
			gStateMachine.status.state 	:= STATE_ERROR;
			gAMS.cmd.abort 				:= TRUE;
		END_IF
	END_IF;

END_ACTION
```

Listed in the project but not available here: Logical/AMS_and_Shunt/CAN/AMS_CAN/Receive/AMS_Receive.st, Logical/AMS_and_Shunt/CAN/AMS_CAN/Receive/Messages/ams_rx_msgs.st, Logical/AMS_and_Shunt/CAN/AMS_CAN/Receive/Messages/orion_rx_msgs.st, Logical/AMS_and_Shunt/CAN/AMS_CAN/Receive/Messages/shunt_rx_msgs.st, Logical/AMS_and_Shunt/CAN/AMS_CAN/Receive/Messages/convertData.st, Logical/AMS_and_Shunt/CAN/AMS_CAN/Receive/functions.st, Logical/Dashboard/Dashboard/Send/Send_Bus.st, Logical/Inverters/CAN/CAN/Send/Send_Bus.st, Logical/Inverters/CAN/CAN/Send/encodeAndSendMessage.st, Logical/Inverters/Control/Control/Mics/convertToKmh.st, Logical/Inverters/Control/Control/Mics/history.st, Logical/Inverters/Control/Control/Mics/frontRearDistribution.st, Logical/Inverters/Control/Control/Mics/accelerationMeasurement.st, Logical/Inverters/Simulation/Simulation, Logical/Libraries/brdkSIM/Types.typ, Logical/Libraries/brdkSIM/Constants.var, Logical/Libraries/brdkSIM/brdkSimInput.c, Logical/Libraries/brdkSIM/brdkSimOutput.c, Logical/Libraries/brdkSTR/brdkSTR.typ, Logical/Libraries/brdkSTR/brdkSTR.var, Logical/Libraries/brdkSTR/brdkSTR.fun, Logical/Libraries/brdkSTR/brdkStrAppendUdintToA.c, Logical/Libraries/brdkSTR/brdkStrAToDint.c, Logical/Libraries/brdkSTR/brdkStrAToUdint.c, Logical/Libraries/brdkSTR/brdkStrCat.c, Logical/Libraries/brdkSTR/brdkStrCatAtChar.c, Logical/Libraries/brdkSTR/brdkStrCharAt.c, Logical/Libraries/brdkSTR/brdkStrCharCount.c, Logical/Libraries/brdkSTR/brdkStrCmp.c, Logical/Libraries/brdkSTR/brdkStrCpy.c, Logical/Libraries/brdkSTR/brdkStrCrc32.c, Logical/Libraries/brdkSTR/brdkStrDintToA.c, Logical/Libraries/brdkSTR/brdkStrFill.c, Logical/Libraries/brdkSTR/brdkStrIndexOf.c, Logical/Libraries/brdkSTR/brdkStrInsertAtPos.c, Logical/Libraries/brdkSTR/brdkStrLen.c, Logical/Libraries/brdkSTR/brdkStrMemCmp.c, Logical/Libraries/brdkSTR/brdkStrMemCpy.c, Logical/Libraries/brdkSTR/brdkStrMemMove.c, Logical/Libraries/brdkSTR/brdkStrMemSet.c, Logical/Libraries/brdkSTR/brdkStrMove.c, Logical/Libraries/brdkSTR/brdkStrNCpy.c, Logical/Libraries/brdkSTR/brdkStrRemove.c, Logical/Libraries/brdkSTR/brdkStrRepeat.c, Logical/Libraries/brdkSTR/brdkStrReplace.c, Logical/Libraries/brdkSTR/brdkStrReverse.c, Logical/Libraries/brdkSTR/brdkStrReverseWords.c, Logical/Libraries/brdkSTR/brdkStrSearch.c, Logical/Libraries/brdkSTR/brdkStrSlice.c, Logical/Libraries/brdkSTR/brdkStrSubStr.c, Logical/Libraries/brdkSTR/brdkStrToDec.c, Logical/Libraries/brdkSTR/brdkStrToHex.c, Logical/Libraries/brdkSTR/brdkStrToLowerCase.c, Logical/Libraries/brdkSTR/brdkStrToUpperCase.c, Logical/Libraries/brdkSTR/brdkStrToUpperCaseWords.c, Logical/Libraries/brdkSTR/brdkStrTrim.c, Logical/Libraries/brdkSTR/brdkStrUdintToA.c, Logical/Libraries/brdkSTR/brdkSTR_func.h, Logical/Libraries/brdkSTR/brdkSTR_func.c, Logical/Libraries/sduVikings/Types.typ, Logical/Libraries/sduVikings/Constants.var, Logical/Libraries/sduVikings/calculateSensorNetOut.st, Logical/Libraries/sduVikings/tractionControl.st, Logical/Libraries/sduVikings/launchProfile.st, Logical/Libraries/sduVikings/torqueLimiter.st, Logical/Libraries/sduVikings/regenerativeBraking.st, Logical/Misc/DataLogging/DataLog/DataLog.st, Logical/Misc/DataLogging/DataLog/Types.typ, Logical/Misc/DataLogging/DataLog/Variables.var, Logical/Misc/DataLogging/DataLog/setup.st, Logical/Misc/DataLogging/globalDataLogging.var, Logical/SC/globalSafetyChain.typ, Logical/SC/SafetyChain/Types.typ, Logical/SC/SafetyChain/Variables.var, Logical/SC/SafetyChain/scUpdate.st, Logical/SC/SafetyChain/scStrings.st, Logical/SC/SafetyChain/eventLog, Logical/SensorNet/globalSensorNet.typ, Logical/SensorNet/globalSensorNet.var
